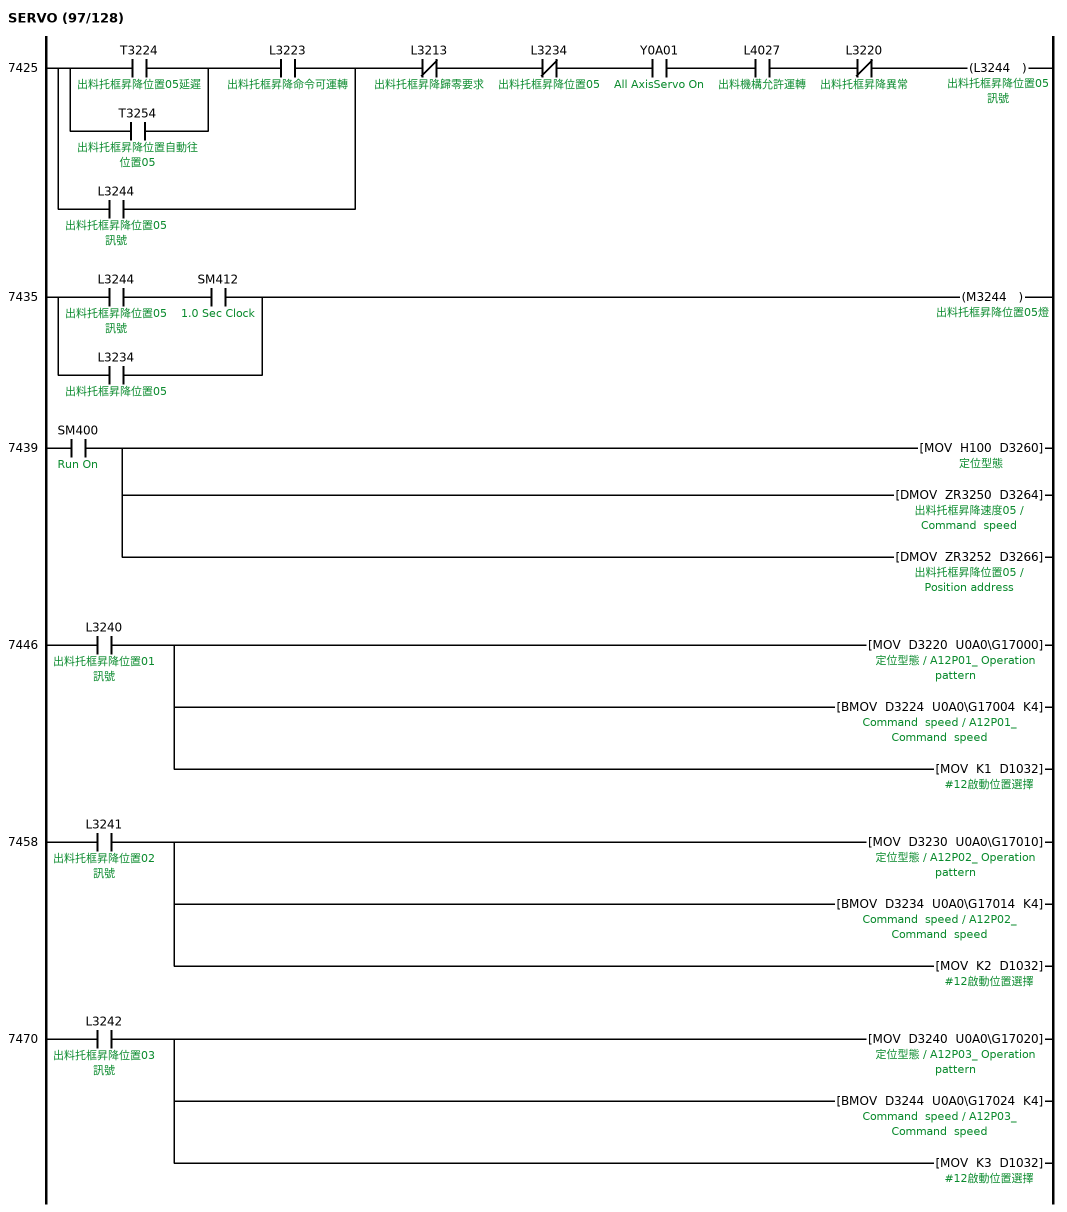
[picture p96: ladder of SERVO, rungs at steps 7425 to 7470]
7425  LD      T3224  ; 出料托框昇降位置05延遲
      OR      T3254  ; 出料托框昇降位置自動往  位置05
      AND     L3223  ; 出料托框昇降命令可運轉
      OR      L3244  ; 出料托框昇降位置05 訊號
      ANI     L3213  ; 出料托框昇降歸零要求
      ANI     L3234  ; 出料托框昇降位置05
      AND     Y0A01  ; All AxisServo On
      AND     L4027  ; 出料機構允許運轉
      ANI     L3220  ; 出料托框昇降異常
      OUT     L3244  ; 出料托框昇降位置05 訊號
7435  LD      L3244  ; 出料托框昇降位置05 訊號
      AND     SM412  ; 1.0 Sec Clock
      OR      L3234  ; 出料托框昇降位置05
      OUT     M3244  ; 出料托框昇降位置05燈
7439  LD      SM400  ; Run On
      MOV     H100 D3260  ; 定位型態
      DMOV    ZR3250 D3264  ; 出料托框昇降速度05 / Command  speed
      DMOV    ZR3252 D3266  ; Position address
7446  LD      L3240  ; 出料托框昇降位置01 訊號
      MOV     D3220 U0A0\G17000  ; A12P01_ Operation pattern
      BMOV    D3224 U0A0\G17004 K4  ; A12P01_ Command  speed
      MOV     K1 D1032  ; #12啟動位置選擇
7458  LD      L3241  ; 出料托框昇降位置02 訊號
      MOV     D3230 U0A0\G17010  ; A12P02_ Operation pattern
      BMOV    D3234 U0A0\G17014 K4  ; A12P02_ Command  speed
      MOV     K2 D1032
7470  LD      L3242  ; 出料托框昇降位置03 訊號
      MOV     D3240 U0A0\G17020  ; A12P03_ Operation pattern
      BMOV    D3244 U0A0\G17024 K4  ; A12P03_ Command  speed
      MOV     K3 D1032
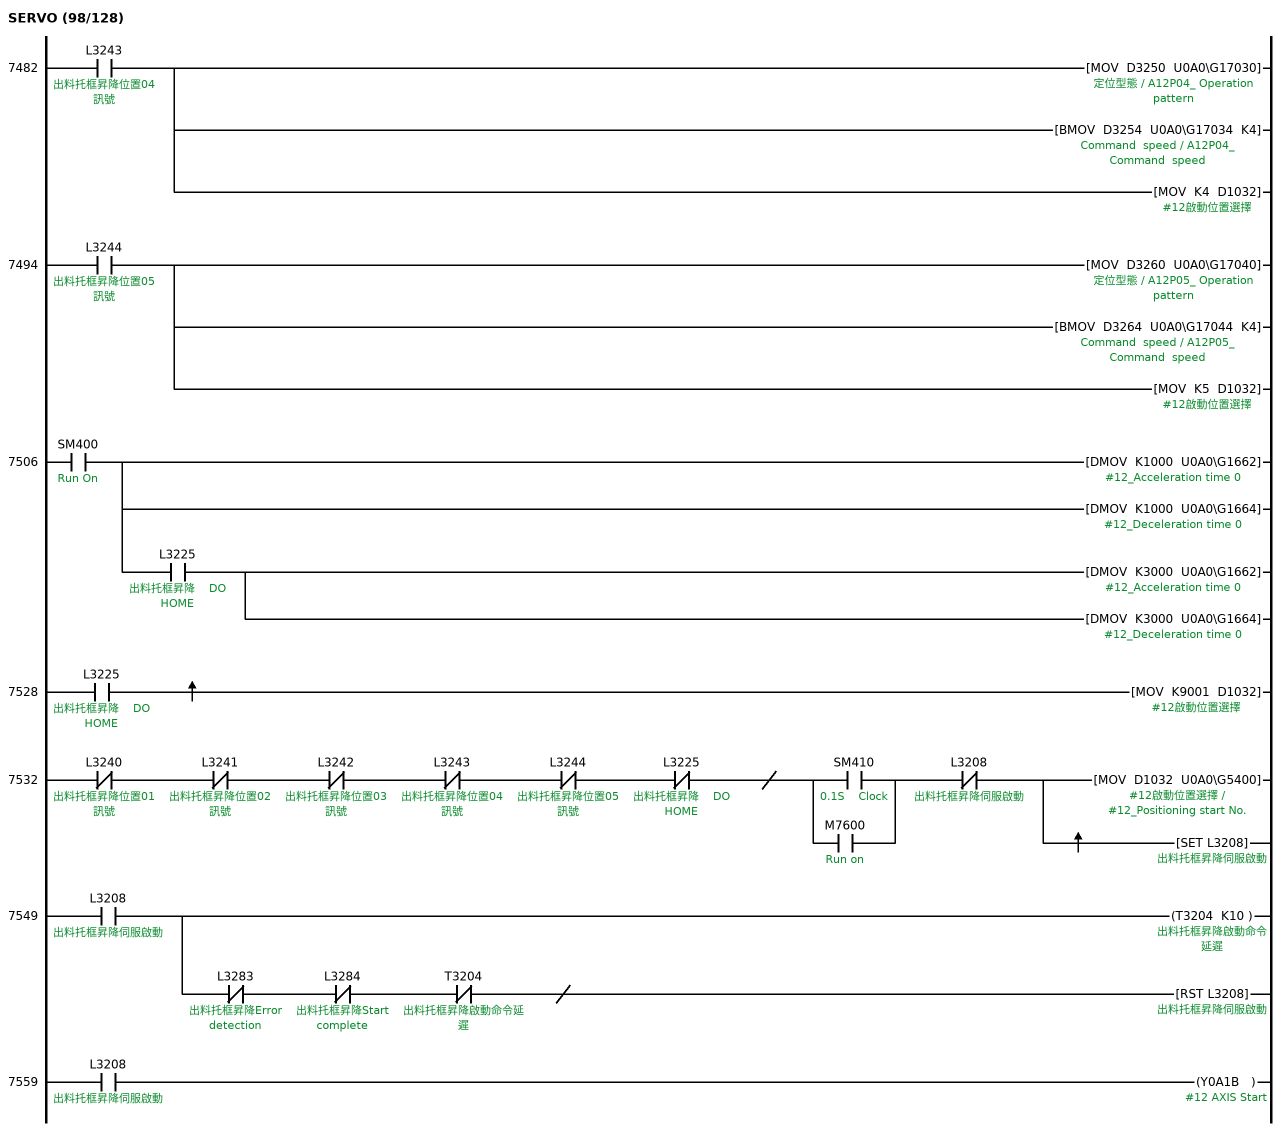
7482  LD      L3243  ; 出料托框昇降位置04 訊號
      MOV     D3250 U0A0\G17030  ; A12P04_ Operation pattern
      BMOV    D3254 U0A0\G17034 K4  ; A12P04_ Command  speed
      MOV     K4 D1032
7494  LD      L3244  ; 出料托框昇降位置05 訊號
      MOV     D3260 U0A0\G17040  ; A12P05_ Operation pattern
      BMOV    D3264 U0A0\G17044 K4  ; A12P05_ Command  speed
      MOV     K5 D1032
7506  LD      SM400  ; Run On
      DMOV    K1000 U0A0\G1662  ; #12_Acceleration time 0
      DMOV    K1000 U0A0\G1664  ; #12_Deceleration time 0
      AND     L3225  ; 出料托框昇降    DO HOME
      DMOV    K3000 U0A0\G1662
      DMOV    K3000 U0A0\G1664
7528  LD      L3225  ; 出料托框昇降    DO HOME
      MEP
      MOV     K9001 D1032
7532  LDI     L3240  ; 出料托框昇降位置01 訊號
      ANI     L3241  ; 出料托框昇降位置02 訊號
      ANI     L3242  ; 出料托框昇降位置03 訊號
      ANI     L3243  ; 出料托框昇降位置04 訊號
      ANI     L3244  ; 出料托框昇降位置05 訊號
      ANI     L3225  ; 出料托框昇降    DO HOME
      INV
      LD      SM410  ; 0.1S    Clock
      OR      M7600  ; Run on
      ANB
      ANI     L3208  ; 出料托框昇降伺服啟動
      MOV     D1032 U0A0\G5400  ; #12_Positioning start No.
      MEP
      SET     L3208  ; 出料托框昇降伺服啟動
7549  LD      L3208  ; 出料托框昇降伺服啟動
      OUT     T3204 K10  ; 出料托框昇降啟動命令延遲
      ANI     L3283  ; 出料托框昇降Error detection
      ANI     L3284  ; 出料托框昇降Start complete
      ANI     T3204  ; 出料托框昇降啟動命令延遲
      INV
      RST     L3208  ; 出料托框昇降伺服啟動
7559  LD      L3208  ; 出料托框昇降伺服啟動
      OUT     Y0A1B  ; #12 AXIS Start
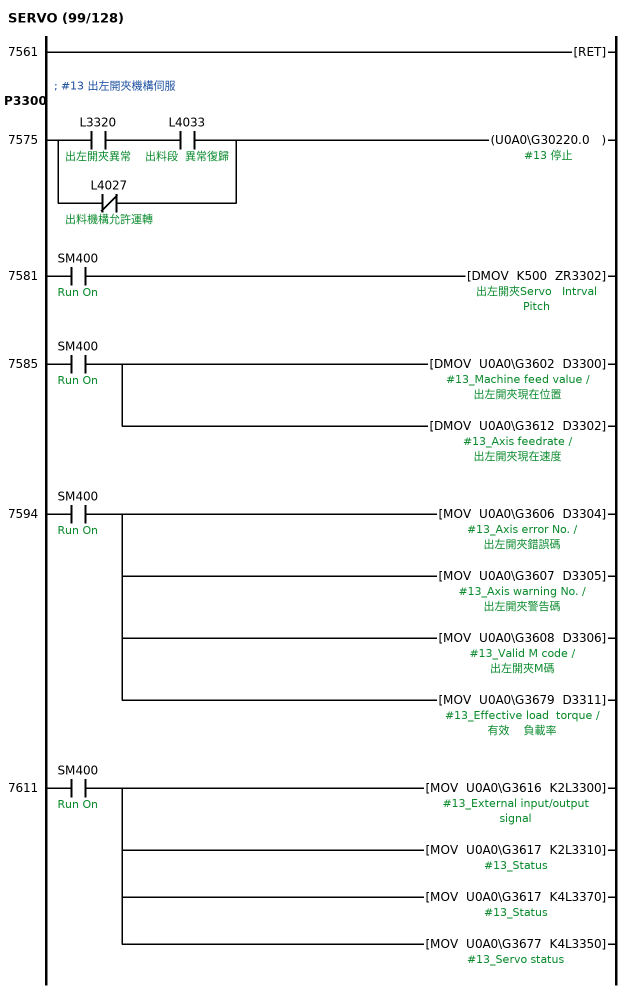
7561  RET
; #13 出左開夾機構伺服
      P3300
7575  LD      L3320  ; 出左開夾異常
      AND     L4033  ; 出料段  異常復歸
      ORI     L4027  ; 出料機構允許運轉
      OUT     U0A0\G30220.0  ; #13 停止
7581  LD      SM400  ; Run On
      DMOV    K500 ZR3302  ; 出左開夾Servo   Intrval Pitch
7585  LD      SM400  ; Run On
      DMOV    U0A0\G3602 D3300  ; #13_Machine feed value / 出左開夾現在位置
      DMOV    U0A0\G3612 D3302  ; #13_Axis feedrate / 出左開夾現在速度
7594  LD      SM400  ; Run On
      MOV     U0A0\G3606 D3304  ; #13_Axis error No. / 出左開夾錯誤碼
      MOV     U0A0\G3607 D3305  ; #13_Axis warning No. / 出左開夾警告碼
      MOV     U0A0\G3608 D3306  ; #13_Valid M code / 出左開夾M碼
      MOV     U0A0\G3679 D3311  ; #13_Effective load  torque / 有效    負載率
7611  LD      SM400  ; Run On
      MOV     U0A0\G3616 K2L3300  ; #13_External input/output signal / 出左開夾    負極限
      MOV     U0A0\G3617 K2L3310  ; #13_Status / 出左開夾速度控制
      MOV     U0A0\G3617 K4L3370  ; 出左開夾速度控制
      MOV     U0A0\G3677 K4L3350  ; #13_Servo status / READY ON
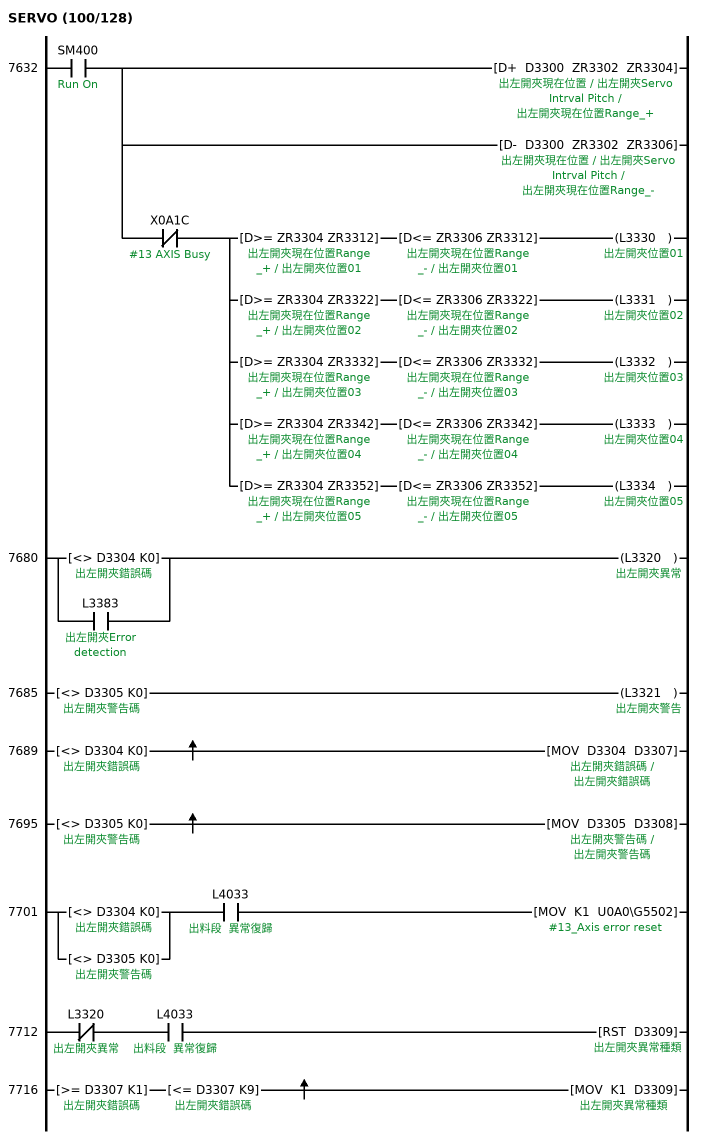
7632  LD      SM400  ; Run On
      D+      D3300 ZR3302 ZR3304  ; 出左開夾現在位置Range_+
      D-      D3300 ZR3302 ZR3306  ; 出左開夾現在位置Range_-
      ANI     X0A1C  ; #13 AXIS Busy
      MPS
      ANDD>=  ZR3304 ZR3312  ; 出左開夾現在位置Range_+ / 出左開夾位置01
      ANDD<=  ZR3306 ZR3312  ; 出左開夾現在位置Range_- / 出左開夾位置01
      OUT     L3330  ; 出左開夾位置01
      MRD
      ANDD>=  ZR3304 ZR3322  ; 出左開夾現在位置Range_+ / 出左開夾位置02
      ANDD<=  ZR3306 ZR3322  ; 出左開夾現在位置Range_- / 出左開夾位置02
      OUT     L3331  ; 出左開夾位置02
      MRD
      ANDD>=  ZR3304 ZR3332  ; 出左開夾現在位置Range_+ / 出左開夾位置03
      ANDD<=  ZR3306 ZR3332  ; 出左開夾現在位置Range_- / 出左開夾位置03
      OUT     L3332  ; 出左開夾位置03
      MRD
      ANDD>=  ZR3304 ZR3342  ; 出左開夾現在位置Range_+ / 出左開夾位置04
      ANDD<=  ZR3306 ZR3342  ; 出左開夾現在位置Range_- / 出左開夾位置04
      OUT     L3333  ; 出左開夾位置04
      MPP
      ANDD>=  ZR3304 ZR3352  ; 出左開夾現在位置Range_+ / 出左開夾位置05
      ANDD<=  ZR3306 ZR3352  ; 出左開夾現在位置Range_- / 出左開夾位置05
      OUT     L3334  ; 出左開夾位置05
7680  LD<>    D3304 K0  ; 出左開夾錯誤碼
      OR      L3383  ; 出左開夾Error detection
      OUT     L3320  ; 出左開夾異常
7685  LD<>    D3305 K0  ; 出左開夾警告碼
      OUT     L3321  ; 出左開夾警告
7689  LD<>    D3304 K0  ; 出左開夾錯誤碼
      MEP
      MOV     D3304 D3307  ; 出左開夾錯誤碼
7695  LD<>    D3305 K0  ; 出左開夾警告碼
      MEP
      MOV     D3305 D3308  ; 出左開夾警告碼
7701  LD<>    D3304 K0  ; 出左開夾錯誤碼
      OR<>    D3305 K0  ; 出左開夾警告碼
      AND     L4033  ; 出料段  異常復歸
      MOV     K1 U0A0\G5502  ; #13_Axis error reset
7712  LDI     L3320  ; 出左開夾異常
      AND     L4033  ; 出料段  異常復歸
      RST     D3309  ; 出左開夾異常種類
7716  LD>=    D3307 K1  ; 出左開夾錯誤碼
      AND<=   D3307 K9  ; 出左開夾錯誤碼
      MEP
      MOV     K1 D3309
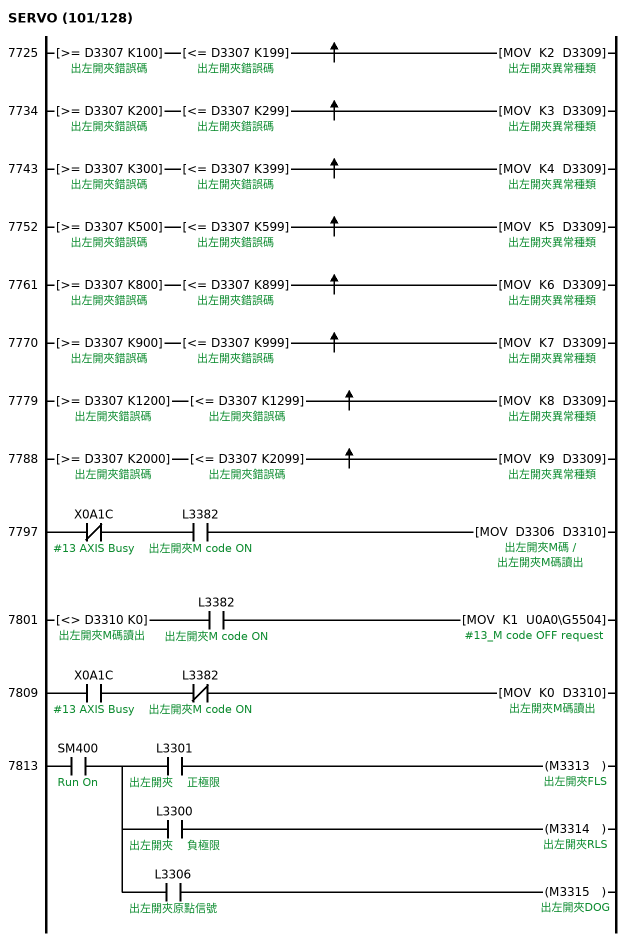
7725  LD>=    D3307 K100  ; 出左開夾錯誤碼
      AND<=   D3307 K199  ; 出左開夾錯誤碼
      MEP
      MOV     K2 D3309
7734  LD>=    D3307 K200  ; 出左開夾錯誤碼
      AND<=   D3307 K299  ; 出左開夾錯誤碼
      MEP
      MOV     K3 D3309
7743  LD>=    D3307 K300  ; 出左開夾錯誤碼
      AND<=   D3307 K399  ; 出左開夾錯誤碼
      MEP
      MOV     K4 D3309
7752  LD>=    D3307 K500  ; 出左開夾錯誤碼
      AND<=   D3307 K599  ; 出左開夾錯誤碼
      MEP
      MOV     K5 D3309
7761  LD>=    D3307 K800  ; 出左開夾錯誤碼
      AND<=   D3307 K899  ; 出左開夾錯誤碼
      MEP
      MOV     K6 D3309
7770  LD>=    D3307 K900  ; 出左開夾錯誤碼
      AND<=   D3307 K999  ; 出左開夾錯誤碼
      MEP
      MOV     K7 D3309
7779  LD>=    D3307 K1200  ; 出左開夾錯誤碼
      AND<=   D3307 K1299  ; 出左開夾錯誤碼
      MEP
      MOV     K8 D3309
7788  LD>=    D3307 K2000  ; 出左開夾錯誤碼
      AND<=   D3307 K2099  ; 出左開夾錯誤碼
      MEP
      MOV     K9 D3309
7797  LDI     X0A1C  ; #13 AXIS Busy
      AND     L3382  ; 出左開夾M code ON
      MOV     D3306 D3310  ; 出左開夾M碼讀出
7801  LD<>    D3310 K0  ; 出左開夾M碼讀出
      AND     L3382  ; 出左開夾M code ON
      MOV     K1 U0A0\G5504  ; #13_M code OFF request
7809  LD      X0A1C  ; #13 AXIS Busy
      ANI     L3382  ; 出左開夾M code ON
      MOV     K0 D3310
7813  LD      SM400  ; Run On
      MPS
      AND     L3301  ; 出左開夾    正極限
      OUT     M3313  ; 出左開夾FLS
      MRD
      AND     L3300  ; 出左開夾    負極限
      OUT     M3314  ; 出左開夾RLS
      MPP
      AND     L3306  ; 出左開夾原點信號
      OUT     M3315  ; 出左開夾DOG
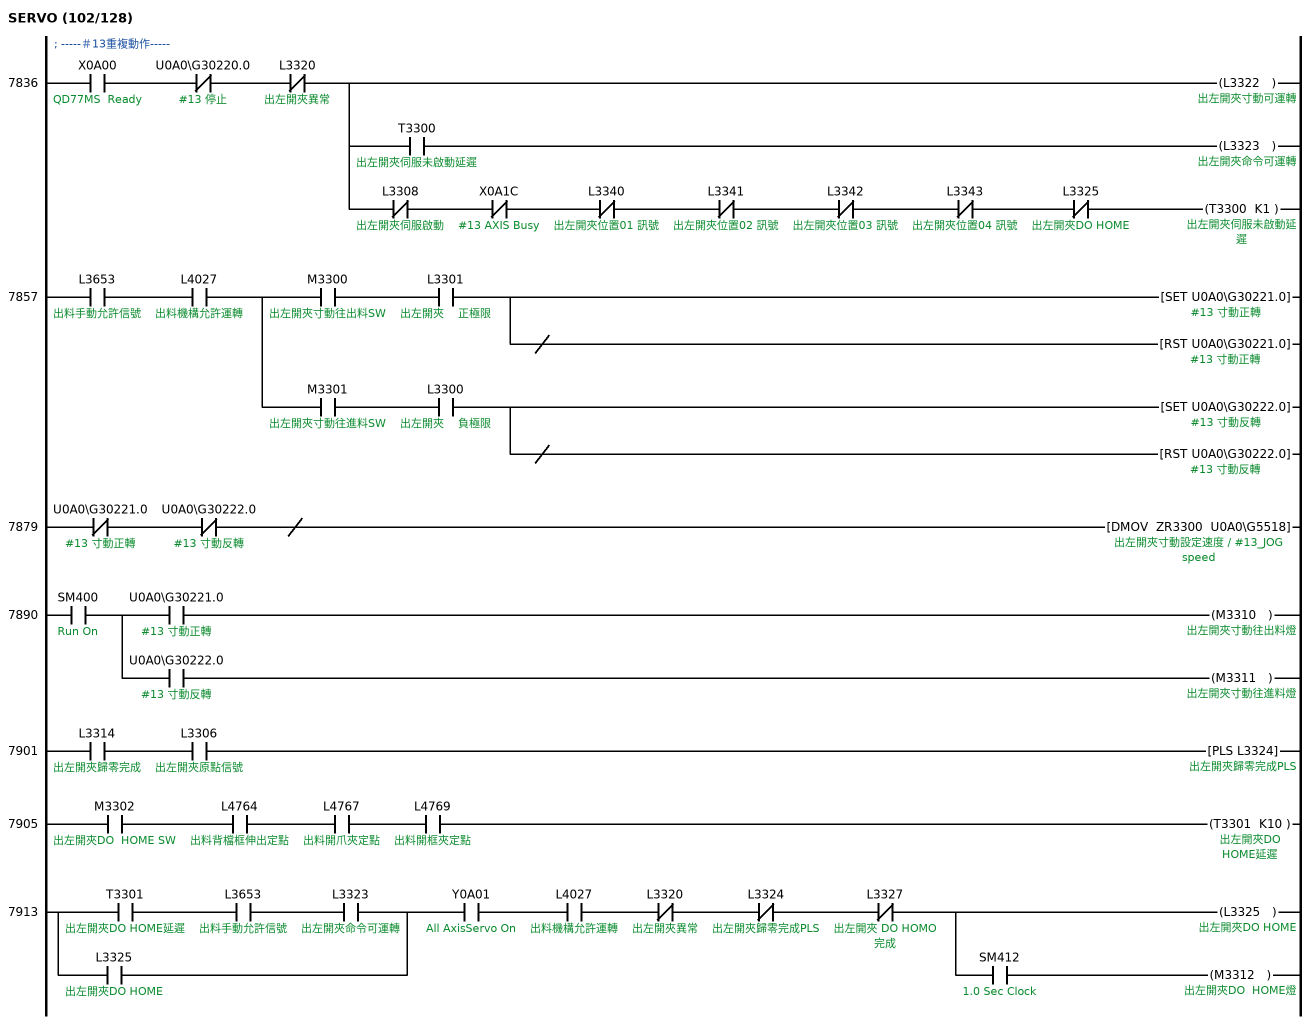
; -----＃13重複動作-----
7836  LD      X0A00  ; QD77MS  Ready
      ANI     U0A0\G30220.0  ; #13 停止
      ANI     L3320  ; 出左開夾異常
      OUT     L3322  ; 出左開夾寸動可運轉
      MPS
      AND     T3300  ; 出左開夾伺服未啟動延遲
      OUT     L3323  ; 出左開夾命令可運轉
      MPP
      ANI     L3308  ; 出左開夾伺服啟動
      ANI     X0A1C  ; #13 AXIS Busy
      ANI     L3340  ; 出左開夾位置01 訊號
      ANI     L3341  ; 出左開夾位置02 訊號
      ANI     L3342  ; 出左開夾位置03 訊號
      ANI     L3343  ; 出左開夾位置04 訊號
      ANI     L3325  ; 出左開夾DO HOME
      OUT     T3300 K1  ; 出左開夾伺服未啟動延遲
7857  LD      L3653  ; 出料手動允許信號
      AND     L4027  ; 出料機構允許運轉
      MPS
      AND     M3300  ; 出左開夾寸動往出料SW
      AND     L3301  ; 出左開夾    正極限
      SET     U0A0\G30221.0  ; #13 寸動正轉
      INV
      RST     U0A0\G30221.0  ; #13 寸動正轉
      MPP
      AND     M3301  ; 出左開夾寸動往進料SW
      AND     L3300  ; 出左開夾    負極限
      SET     U0A0\G30222.0  ; #13 寸動反轉
      INV
      RST     U0A0\G30222.0  ; #13 寸動反轉
7879  LDI     U0A0\G30221.0  ; #13 寸動正轉
      ANI     U0A0\G30222.0  ; #13 寸動反轉
      INV
      DMOV    ZR3300 U0A0\G5518  ; 出左開夾寸動設定速度 / #13_JOG     speed
7890  LD      SM400  ; Run On
      MPS
      AND     U0A0\G30221.0  ; #13 寸動正轉
      OUT     M3310  ; 出左開夾寸動往出料燈
      MPP
      AND     U0A0\G30222.0  ; #13 寸動反轉
      OUT     M3311  ; 出左開夾寸動往進料燈
7901  LD      L3314  ; 出左開夾歸零完成
      AND     L3306  ; 出左開夾原點信號
      PLS     L3324  ; 出左開夾歸零完成PLS
7905  LD      M3302  ; 出左開夾DO  HOME SW
      AND     L4764  ; 出料背檔框伸出定點
      AND     L4767  ; 出料開爪夾定點
      AND     L4769  ; 出料開框夾定點
      OUT     T3301 K10  ; 出左開夾DO HOME延遲
7913  LD      T3301  ; 出左開夾DO HOME延遲
      AND     L3653  ; 出料手動允許信號
      AND     L3323  ; 出左開夾命令可運轉
      OR      L3325  ; 出左開夾DO HOME
      AND     Y0A01  ; All AxisServo On
      AND     L4027  ; 出料機構允許運轉
      ANI     L3320  ; 出左開夾異常
      ANI     L3324  ; 出左開夾歸零完成PLS
      ANI     L3327  ; 出左開夾 DO HOMO 完成
      OUT     L3325  ; 出左開夾DO HOME
      AND     SM412  ; 1.0 Sec Clock
      OUT     M3312  ; 出左開夾DO  HOME燈
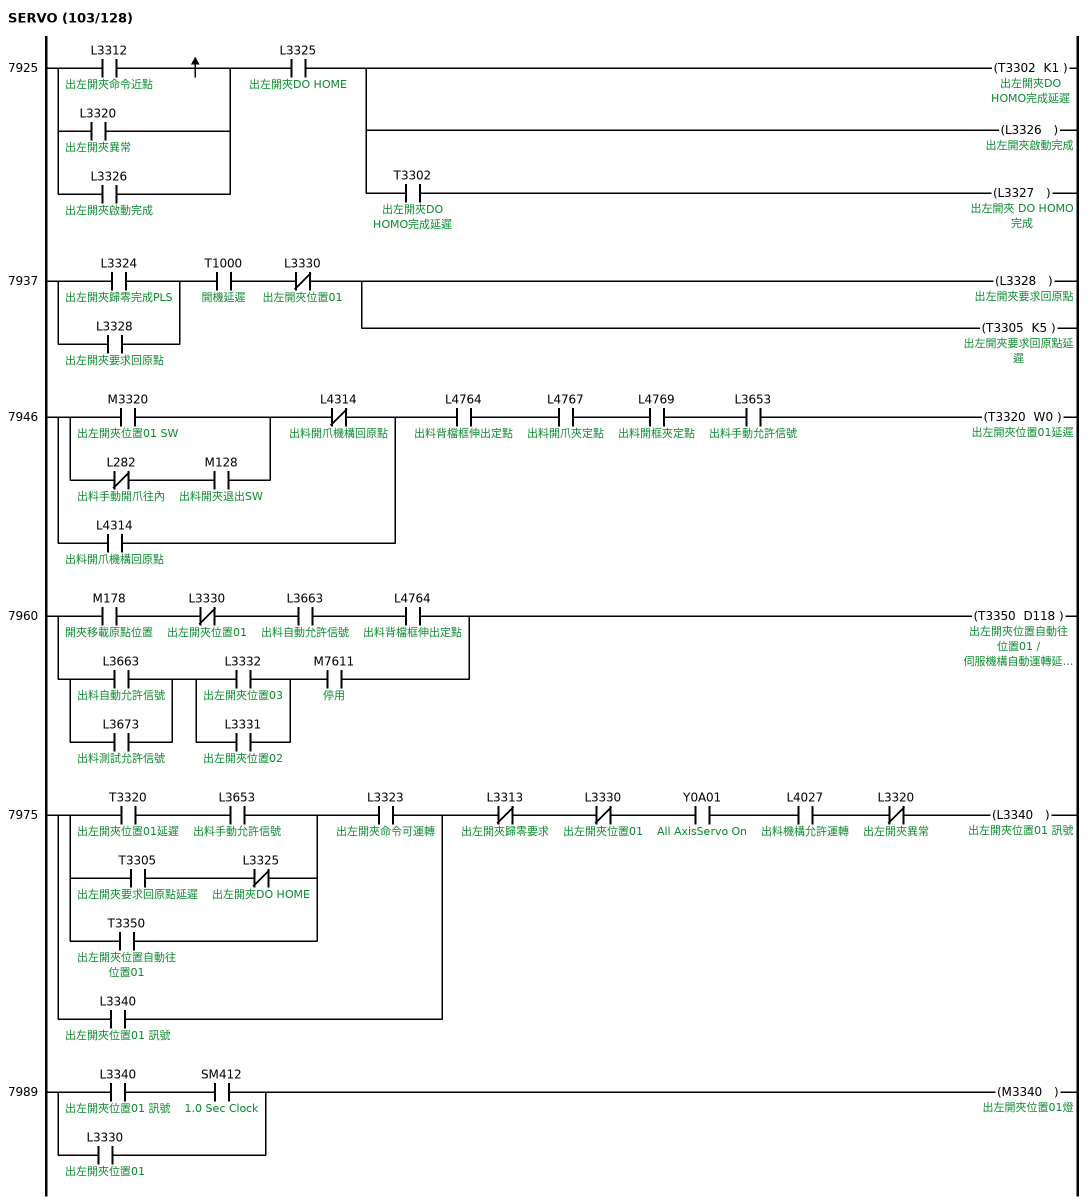
7925  LD      L3312  ; 出左開夾命令近點
      MEP
      OR      L3320  ; 出左開夾異常
      OR      L3326  ; 出左開夾啟動完成
      AND     L3325  ; 出左開夾DO HOME
      OUT     T3302 K1  ; 出左開夾DO HOMO完成延遲
      OUT     L3326  ; 出左開夾啟動完成
      AND     T3302  ; 出左開夾DO HOMO完成延遲
      OUT     L3327  ; 出左開夾 DO HOMO 完成
7937  LD      L3324  ; 出左開夾歸零完成PLS
      OR      L3328  ; 出左開夾要求回原點
      AND     T1000  ; 開機延遲
      ANI     L3330  ; 出左開夾位置01
      OUT     L3328  ; 出左開夾要求回原點
      OUT     T3305 K5  ; 出左開夾要求回原點延遲
7946  LD      M3320  ; 出左開夾位置01 SW
      LDI     L282  ; 出料手動開爪往內
      AND     M128  ; 出料開夾退出SW
      ORB
      ANI     L4314  ; 出料開爪機構回原點
      OR      L4314  ; 出料開爪機構回原點
      AND     L4764  ; 出料背檔框伸出定點
      AND     L4767  ; 出料開爪夾定點
      AND     L4769  ; 出料開框夾定點
      AND     L3653  ; 出料手動允許信號
      OUT     T3320 W0  ; 出左開夾位置01延遲
7960  LD      M178  ; 開夾移載原點位置
      ANI     L3330  ; 出左開夾位置01
      AND     L3663  ; 出料自動允許信號
      AND     L4764  ; 出料背檔框伸出定點
      LD      L3663  ; 出料自動允許信號
      OR      L3673  ; 出料測試允許信號
      LD      L3332  ; 出左開夾位置03
      OR      L3331  ; 出左開夾位置02
      ANB
      AND     M7611  ; 停用
      ORB
      OUT     T3350 D118  ; 出左開夾位置自動往  位置01 / 伺服機構自動運轉延遲時間
7975  LD      T3320  ; 出左開夾位置01延遲
      AND     L3653  ; 出料手動允許信號
      LD      T3305  ; 出左開夾要求回原點延遲
      ANI     L3325  ; 出左開夾DO HOME
      ORB
      OR      T3350  ; 出左開夾位置自動往  位置01
      AND     L3323  ; 出左開夾命令可運轉
      OR      L3340  ; 出左開夾位置01 訊號
      ANI     L3313  ; 出左開夾歸零要求
      ANI     L3330  ; 出左開夾位置01
      AND     Y0A01  ; All AxisServo On
      AND     L4027  ; 出料機構允許運轉
      ANI     L3320  ; 出左開夾異常
      OUT     L3340  ; 出左開夾位置01 訊號
7989  LD      L3340  ; 出左開夾位置01 訊號
      AND     SM412  ; 1.0 Sec Clock
      OR      L3330  ; 出左開夾位置01
      OUT     M3340  ; 出左開夾位置01燈
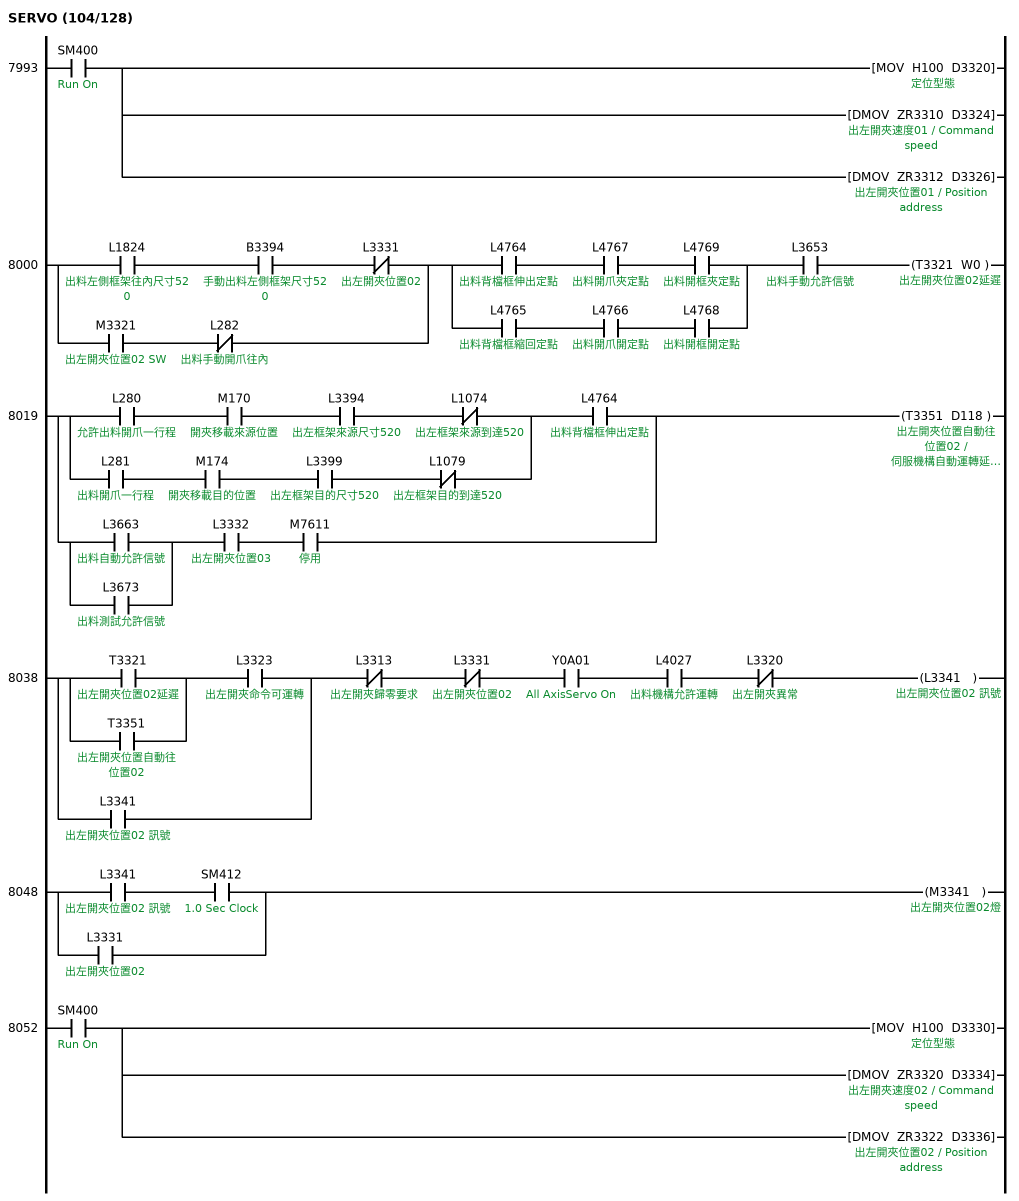
7993  LD      SM400  ; Run On
      MOV     H100 D3320  ; 定位型態
      DMOV    ZR3310 D3324  ; 出左開夾速度01 / Command  speed
      DMOV    ZR3312 D3326  ; Position address
8000  LD      L1824  ; 出料左側框架往內尺寸520
      AND     B3394  ; 手動出料左側框架尺寸520
      ANI     L3331  ; 出左開夾位置02
      LD      M3321  ; 出左開夾位置02 SW
      ANI     L282  ; 出料手動開爪往內
      ORB
      LD      L4764  ; 出料背檔框伸出定點
      AND     L4767  ; 出料開爪夾定點
      AND     L4769  ; 出料開框夾定點
      LD      L4765  ; 出料背檔框縮回定點
      AND     L4766  ; 出料開爪開定點
      AND     L4768  ; 出料開框開定點
      ORB
      ANB
      AND     L3653  ; 出料手動允許信號
      OUT     T3321 W0  ; 出左開夾位置02延遲
8019  LD      L280  ; 允許出料開爪一行程
      AND     M170  ; 開夾移載來源位置
      AND     L3394  ; 出左框架來源尺寸520
      ANI     L1074  ; 出左框架來源到達520
      LD      L281  ; 出料開爪一行程
      AND     M174  ; 開夾移載目的位置
      AND     L3399  ; 出左框架目的尺寸520
      ANI     L1079  ; 出左框架目的到達520
      ORB
      AND     L4764  ; 出料背檔框伸出定點
      LD      L3663  ; 出料自動允許信號
      OR      L3673  ; 出料測試允許信號
      AND     L3332  ; 出左開夾位置03
      AND     M7611  ; 停用
      ORB
      OUT     T3351 D118  ; 出左開夾位置自動往  位置02 / 伺服機構自動運轉延遲時間
8038  LD      T3321  ; 出左開夾位置02延遲
      OR      T3351  ; 出左開夾位置自動往  位置02
      AND     L3323  ; 出左開夾命令可運轉
      OR      L3341  ; 出左開夾位置02 訊號
      ANI     L3313  ; 出左開夾歸零要求
      ANI     L3331  ; 出左開夾位置02
      AND     Y0A01  ; All AxisServo On
      AND     L4027  ; 出料機構允許運轉
      ANI     L3320  ; 出左開夾異常
      OUT     L3341  ; 出左開夾位置02 訊號
8048  LD      L3341  ; 出左開夾位置02 訊號
      AND     SM412  ; 1.0 Sec Clock
      OR      L3331  ; 出左開夾位置02
      OUT     M3341  ; 出左開夾位置02燈
8052  LD      SM400  ; Run On
      MOV     H100 D3330  ; 定位型態
      DMOV    ZR3320 D3334  ; 出左開夾速度02 / Command  speed
      DMOV    ZR3322 D3336  ; Position address
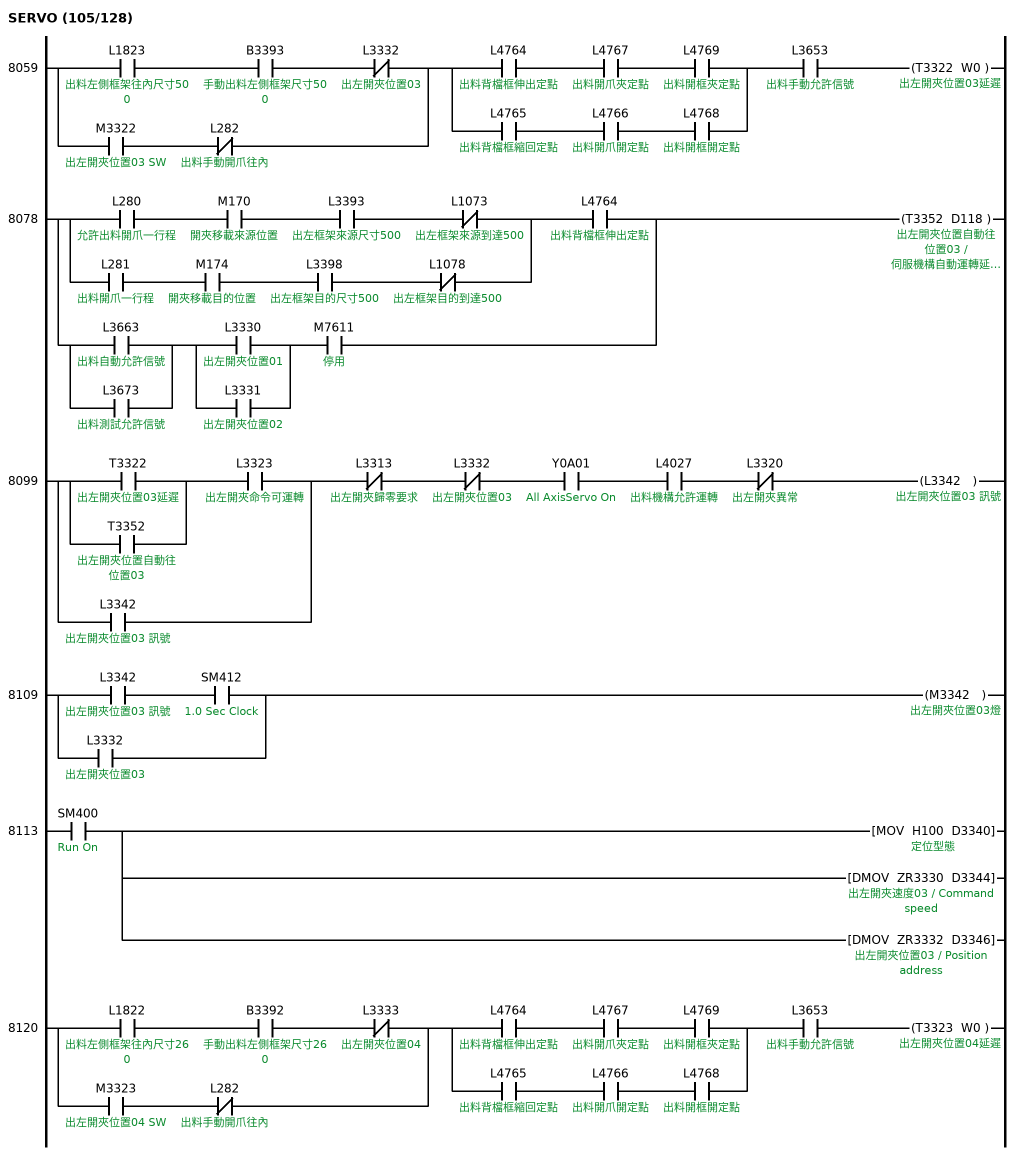
8059  LD      L1823  ; 出料左側框架往內尺寸500
      AND     B3393  ; 手動出料左側框架尺寸500
      ANI     L3332  ; 出左開夾位置03
      LD      M3322  ; 出左開夾位置03 SW
      ANI     L282  ; 出料手動開爪往內
      ORB
      LD      L4764  ; 出料背檔框伸出定點
      AND     L4767  ; 出料開爪夾定點
      AND     L4769  ; 出料開框夾定點
      LD      L4765  ; 出料背檔框縮回定點
      AND     L4766  ; 出料開爪開定點
      AND     L4768  ; 出料開框開定點
      ORB
      ANB
      AND     L3653  ; 出料手動允許信號
      OUT     T3322 W0  ; 出左開夾位置03延遲
8078  LD      L280  ; 允許出料開爪一行程
      AND     M170  ; 開夾移載來源位置
      AND     L3393  ; 出左框架來源尺寸500
      ANI     L1073  ; 出左框架來源到達500
      LD      L281  ; 出料開爪一行程
      AND     M174  ; 開夾移載目的位置
      AND     L3398  ; 出左框架目的尺寸500
      ANI     L1078  ; 出左框架目的到達500
      ORB
      AND     L4764  ; 出料背檔框伸出定點
      LD      L3663  ; 出料自動允許信號
      OR      L3673  ; 出料測試允許信號
      LD      L3330  ; 出左開夾位置01
      OR      L3331  ; 出左開夾位置02
      ANB
      AND     M7611  ; 停用
      ORB
      OUT     T3352 D118  ; 出左開夾位置自動往  位置03 / 伺服機構自動運轉延遲時間
8099  LD      T3322  ; 出左開夾位置03延遲
      OR      T3352  ; 出左開夾位置自動往  位置03
      AND     L3323  ; 出左開夾命令可運轉
      OR      L3342  ; 出左開夾位置03 訊號
      ANI     L3313  ; 出左開夾歸零要求
      ANI     L3332  ; 出左開夾位置03
      AND     Y0A01  ; All AxisServo On
      AND     L4027  ; 出料機構允許運轉
      ANI     L3320  ; 出左開夾異常
      OUT     L3342  ; 出左開夾位置03 訊號
8109  LD      L3342  ; 出左開夾位置03 訊號
      AND     SM412  ; 1.0 Sec Clock
      OR      L3332  ; 出左開夾位置03
      OUT     M3342  ; 出左開夾位置03燈
8113  LD      SM400  ; Run On
      MOV     H100 D3340  ; 定位型態
      DMOV    ZR3330 D3344  ; 出左開夾速度03 / Command  speed
      DMOV    ZR3332 D3346  ; Position address
8120  LD      L1822  ; 出料左側框架往內尺寸260
      AND     B3392  ; 手動出料左側框架尺寸260
      ANI     L3333  ; 出左開夾位置04
      LD      M3323  ; 出左開夾位置04 SW
      ANI     L282  ; 出料手動開爪往內
      ORB
      LD      L4764  ; 出料背檔框伸出定點
      AND     L4767  ; 出料開爪夾定點
      AND     L4769  ; 出料開框夾定點
      LD      L4765  ; 出料背檔框縮回定點
      AND     L4766  ; 出料開爪開定點
      AND     L4768  ; 出料開框開定點
      ORB
      ANB
      AND     L3653  ; 出料手動允許信號
      OUT     T3323 W0  ; 出左開夾位置04延遲
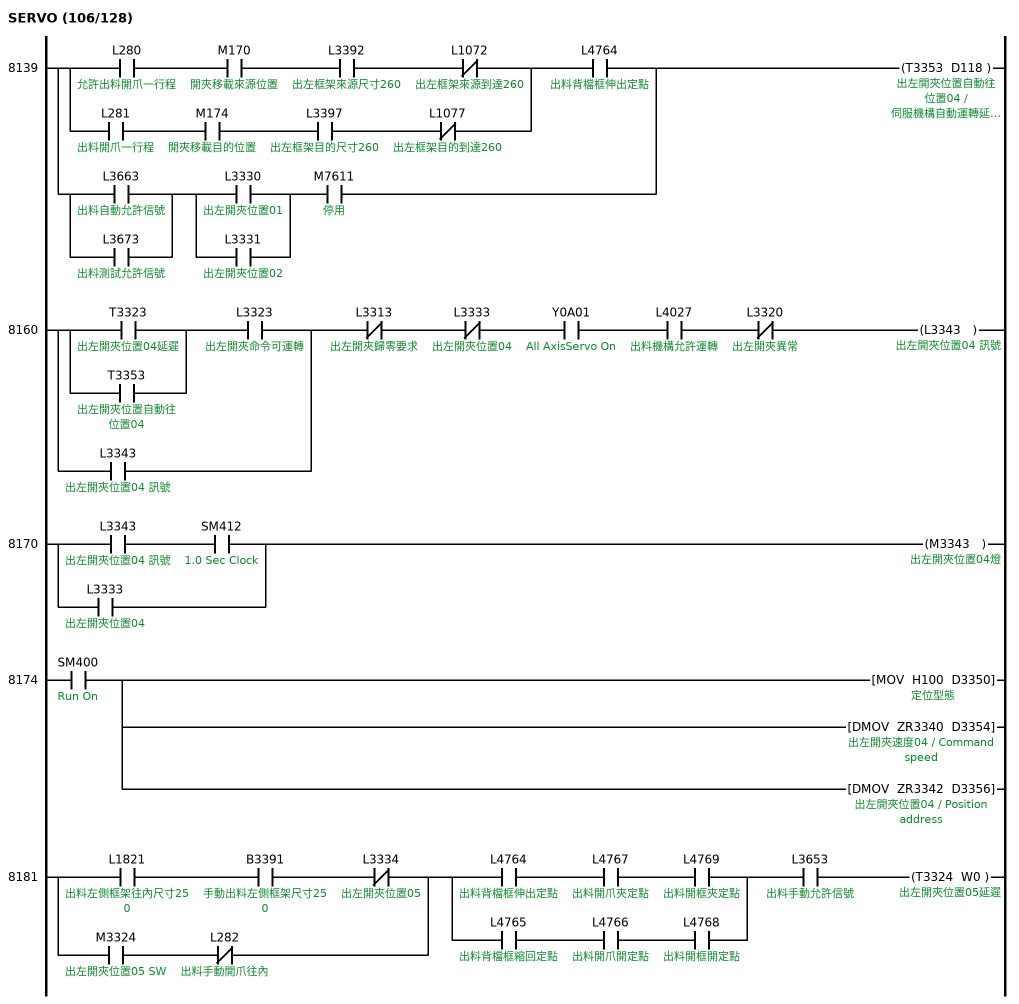
8139  LD      L280  ; 允許出料開爪一行程
      AND     M170  ; 開夾移載來源位置
      AND     L3392  ; 出左框架來源尺寸260
      ANI     L1072  ; 出左框架來源到達260
      LD      L281  ; 出料開爪一行程
      AND     M174  ; 開夾移載目的位置
      AND     L3397  ; 出左框架目的尺寸260
      ANI     L1077  ; 出左框架目的到達260
      ORB
      AND     L4764  ; 出料背檔框伸出定點
      LD      L3663  ; 出料自動允許信號
      OR      L3673  ; 出料測試允許信號
      LD      L3330  ; 出左開夾位置01
      OR      L3331  ; 出左開夾位置02
      ANB
      AND     M7611  ; 停用
      ORB
      OUT     T3353 D118  ; 出左開夾位置自動往  位置04 / 伺服機構自動運轉延遲時間
8160  LD      T3323  ; 出左開夾位置04延遲
      OR      T3353  ; 出左開夾位置自動往  位置04
      AND     L3323  ; 出左開夾命令可運轉
      OR      L3343  ; 出左開夾位置04 訊號
      ANI     L3313  ; 出左開夾歸零要求
      ANI     L3333  ; 出左開夾位置04
      AND     Y0A01  ; All AxisServo On
      AND     L4027  ; 出料機構允許運轉
      ANI     L3320  ; 出左開夾異常
      OUT     L3343  ; 出左開夾位置04 訊號
8170  LD      L3343  ; 出左開夾位置04 訊號
      AND     SM412  ; 1.0 Sec Clock
      OR      L3333  ; 出左開夾位置04
      OUT     M3343  ; 出左開夾位置04燈
8174  LD      SM400  ; Run On
      MOV     H100 D3350  ; 定位型態
      DMOV    ZR3340 D3354  ; 出左開夾速度04 / Command  speed
      DMOV    ZR3342 D3356  ; Position address
8181  LD      L1821  ; 出料左側框架往內尺寸250
      AND     B3391  ; 手動出料左側框架尺寸250
      ANI     L3334  ; 出左開夾位置05
      LD      M3324  ; 出左開夾位置05 SW
      ANI     L282  ; 出料手動開爪往內
      ORB
      LD      L4764  ; 出料背檔框伸出定點
      AND     L4767  ; 出料開爪夾定點
      AND     L4769  ; 出料開框夾定點
      LD      L4765  ; 出料背檔框縮回定點
      AND     L4766  ; 出料開爪開定點
      AND     L4768  ; 出料開框開定點
      ORB
      ANB
      AND     L3653  ; 出料手動允許信號
      OUT     T3324 W0  ; 出左開夾位置05延遲
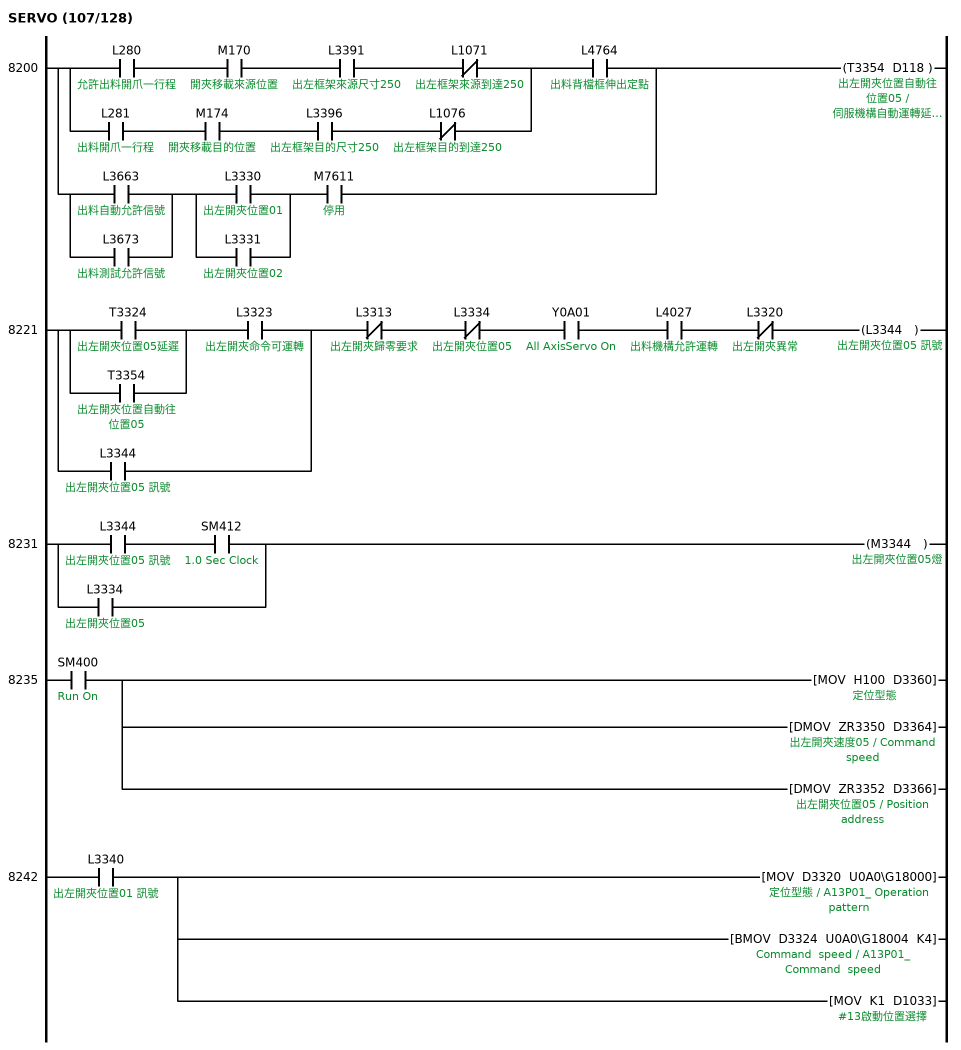
8200  LD      L280  ; 允許出料開爪一行程
      AND     M170  ; 開夾移載來源位置
      AND     L3391  ; 出左框架來源尺寸250
      ANI     L1071  ; 出左框架來源到達250
      LD      L281  ; 出料開爪一行程
      AND     M174  ; 開夾移載目的位置
      AND     L3396  ; 出左框架目的尺寸250
      ANI     L1076  ; 出左框架目的到達250
      ORB
      AND     L4764  ; 出料背檔框伸出定點
      LD      L3663  ; 出料自動允許信號
      OR      L3673  ; 出料測試允許信號
      LD      L3330  ; 出左開夾位置01
      OR      L3331  ; 出左開夾位置02
      ANB
      AND     M7611  ; 停用
      ORB
      OUT     T3354 D118  ; 出左開夾位置自動往  位置05 / 伺服機構自動運轉延遲時間
8221  LD      T3324  ; 出左開夾位置05延遲
      OR      T3354  ; 出左開夾位置自動往  位置05
      AND     L3323  ; 出左開夾命令可運轉
      OR      L3344  ; 出左開夾位置05 訊號
      ANI     L3313  ; 出左開夾歸零要求
      ANI     L3334  ; 出左開夾位置05
      AND     Y0A01  ; All AxisServo On
      AND     L4027  ; 出料機構允許運轉
      ANI     L3320  ; 出左開夾異常
      OUT     L3344  ; 出左開夾位置05 訊號
8231  LD      L3344  ; 出左開夾位置05 訊號
      AND     SM412  ; 1.0 Sec Clock
      OR      L3334  ; 出左開夾位置05
      OUT     M3344  ; 出左開夾位置05燈
8235  LD      SM400  ; Run On
      MOV     H100 D3360  ; 定位型態
      DMOV    ZR3350 D3364  ; 出左開夾速度05 / Command  speed
      DMOV    ZR3352 D3366  ; Position address
8242  LD      L3340  ; 出左開夾位置01 訊號
      MOV     D3320 U0A0\G18000  ; A13P01_ Operation pattern
      BMOV    D3324 U0A0\G18004 K4  ; A13P01_ Command  speed
      MOV     K1 D1033  ; #13啟動位置選擇
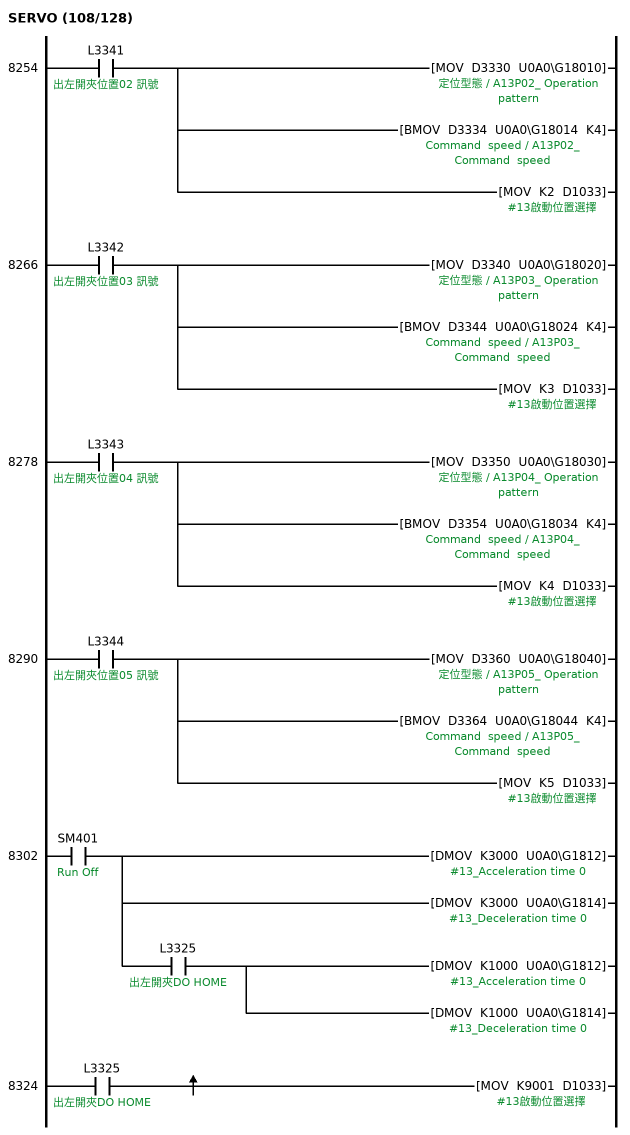
8254  LD      L3341  ; 出左開夾位置02 訊號
      MOV     D3330 U0A0\G18010  ; A13P02_ Operation pattern
      BMOV    D3334 U0A0\G18014 K4  ; A13P02_ Command  speed
      MOV     K2 D1033
8266  LD      L3342  ; 出左開夾位置03 訊號
      MOV     D3340 U0A0\G18020  ; A13P03_ Operation pattern
      BMOV    D3344 U0A0\G18024 K4  ; A13P03_ Command  speed
      MOV     K3 D1033
8278  LD      L3343  ; 出左開夾位置04 訊號
      MOV     D3350 U0A0\G18030  ; A13P04_ Operation pattern
      BMOV    D3354 U0A0\G18034 K4  ; A13P04_ Command  speed
      MOV     K4 D1033
8290  LD      L3344  ; 出左開夾位置05 訊號
      MOV     D3360 U0A0\G18040  ; A13P05_ Operation pattern
      BMOV    D3364 U0A0\G18044 K4  ; A13P05_ Command  speed
      MOV     K5 D1033
8302  LD      SM401  ; Run Off
      DMOV    K3000 U0A0\G1812  ; #13_Acceleration time 0
      DMOV    K3000 U0A0\G1814  ; #13_Deceleration time 0
      AND     L3325  ; 出左開夾DO HOME
      DMOV    K1000 U0A0\G1812
      DMOV    K1000 U0A0\G1814
8324  LD      L3325  ; 出左開夾DO HOME
      MEP
      MOV     K9001 D1033
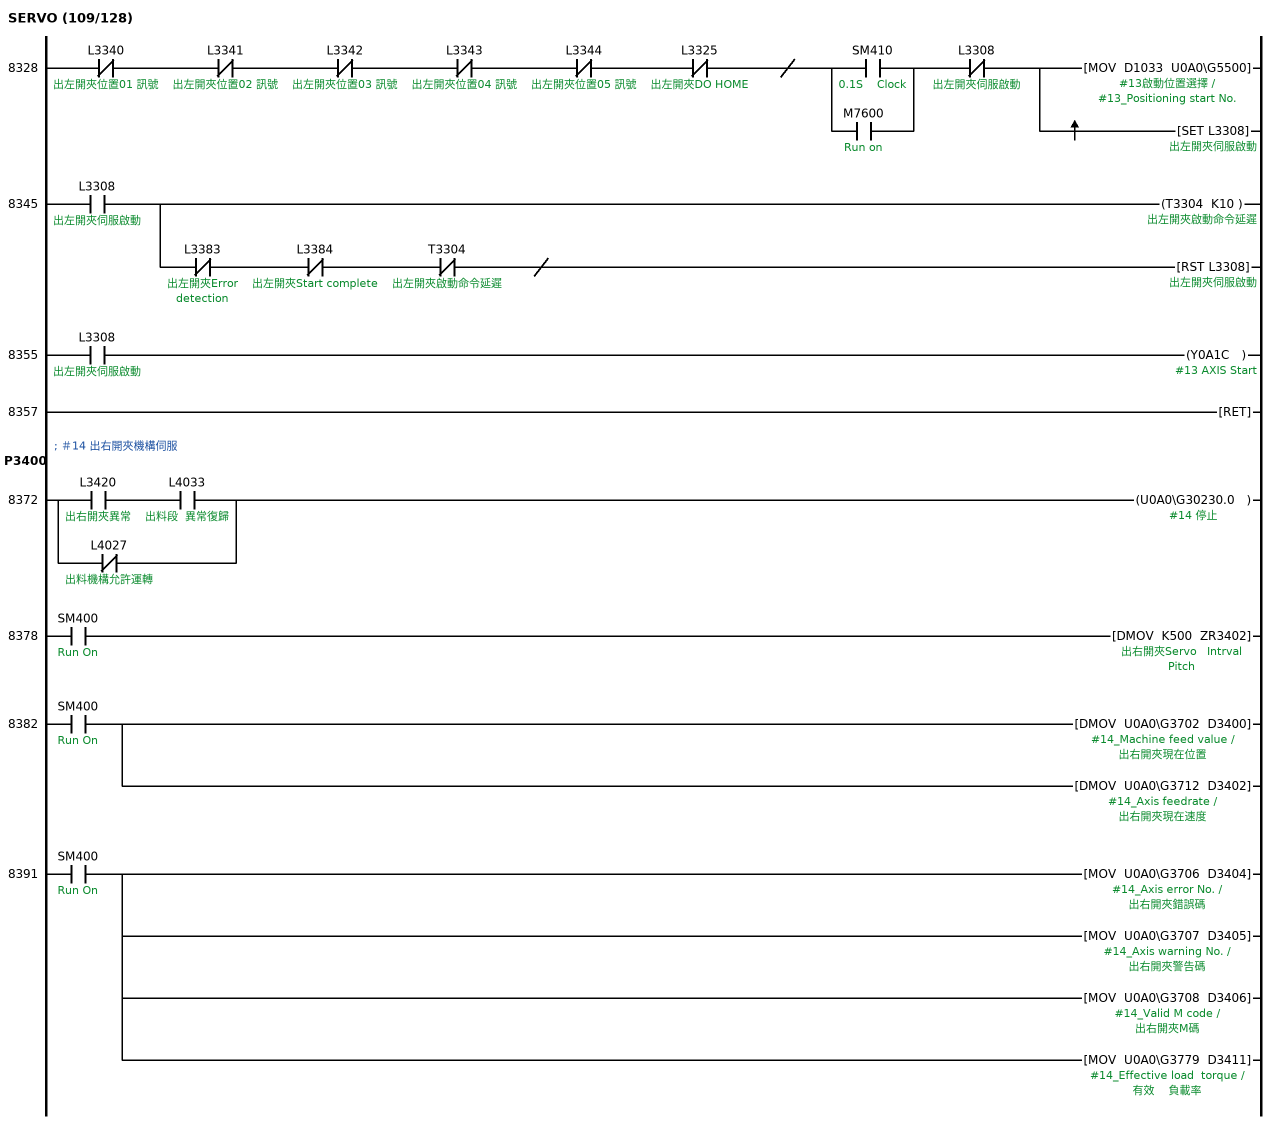
8328  LDI     L3340  ; 出左開夾位置01 訊號
      ANI     L3341  ; 出左開夾位置02 訊號
      ANI     L3342  ; 出左開夾位置03 訊號
      ANI     L3343  ; 出左開夾位置04 訊號
      ANI     L3344  ; 出左開夾位置05 訊號
      ANI     L3325  ; 出左開夾DO HOME
      INV
      LD      SM410  ; 0.1S    Clock
      OR      M7600  ; Run on
      ANB
      ANI     L3308  ; 出左開夾伺服啟動
      MOV     D1033 U0A0\G5500  ; #13_Positioning start No.
      MEP
      SET     L3308  ; 出左開夾伺服啟動
8345  LD      L3308  ; 出左開夾伺服啟動
      OUT     T3304 K10  ; 出左開夾啟動命令延遲
      ANI     L3383  ; 出左開夾Error detection
      ANI     L3384  ; 出左開夾Start complete
      ANI     T3304  ; 出左開夾啟動命令延遲
      INV
      RST     L3308  ; 出左開夾伺服啟動
8355  LD      L3308  ; 出左開夾伺服啟動
      OUT     Y0A1C  ; #13 AXIS Start
8357  RET
; ＃14 出右開夾機構伺服
      P3400
8372  LD      L3420  ; 出右開夾異常
      AND     L4033  ; 出料段  異常復歸
      ORI     L4027  ; 出料機構允許運轉
      OUT     U0A0\G30230.0  ; #14 停止
8378  LD      SM400  ; Run On
      DMOV    K500 ZR3402  ; 出右開夾Servo   Intrval Pitch
8382  LD      SM400  ; Run On
      DMOV    U0A0\G3702 D3400  ; #14_Machine feed value / 出右開夾現在位置
      DMOV    U0A0\G3712 D3402  ; #14_Axis feedrate / 出右開夾現在速度
8391  LD      SM400  ; Run On
      MOV     U0A0\G3706 D3404  ; #14_Axis error No. / 出右開夾錯誤碼
      MOV     U0A0\G3707 D3405  ; #14_Axis warning No. / 出右開夾警告碼
      MOV     U0A0\G3708 D3406  ; #14_Valid M code / 出右開夾M碼
      MOV     U0A0\G3779 D3411  ; #14_Effective load  torque / 有效    負載率
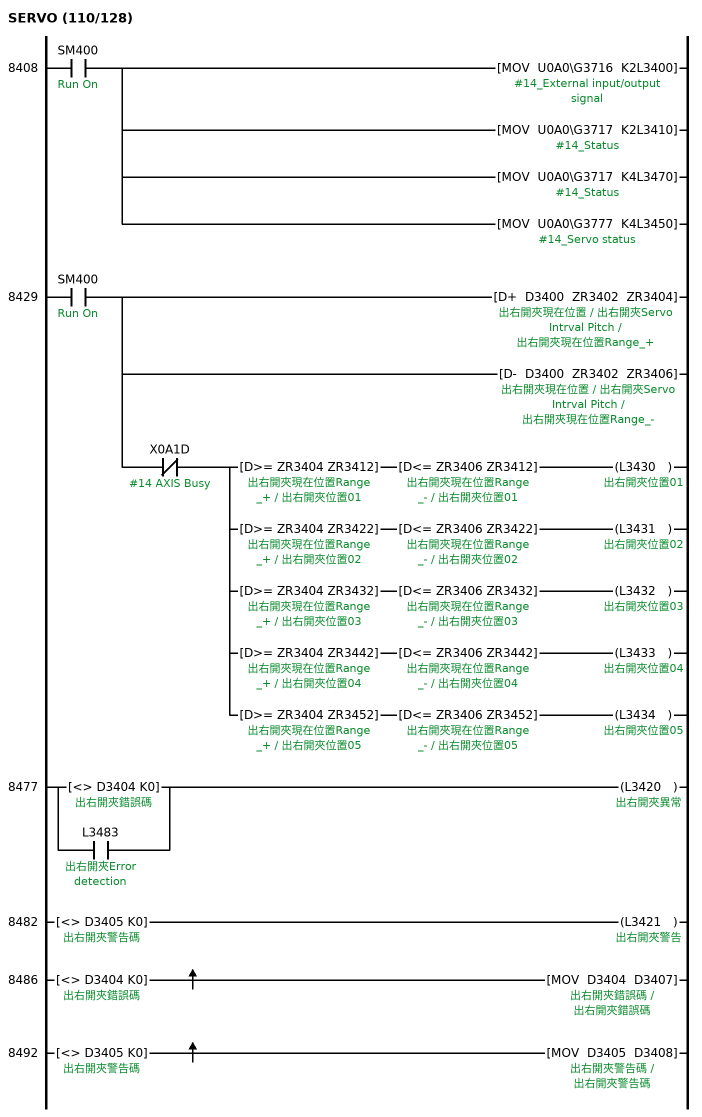
8408  LD      SM400  ; Run On
      MOV     U0A0\G3716 K2L3400  ; #14_External input/output signal / 出右開夾    負極限
      MOV     U0A0\G3717 K2L3410  ; #14_Status / 出右開夾速度控制
      MOV     U0A0\G3717 K4L3470  ; 出右開夾速度控制
      MOV     U0A0\G3777 K4L3450  ; #14_Servo status / READY ON
8429  LD      SM400  ; Run On
      D+      D3400 ZR3402 ZR3404  ; 出右開夾現在位置Range_+
      D-      D3400 ZR3402 ZR3406  ; 出右開夾現在位置Range_-
      ANI     X0A1D  ; #14 AXIS Busy
      MPS
      ANDD>=  ZR3404 ZR3412  ; 出右開夾現在位置Range_+ / 出右開夾位置01
      ANDD<=  ZR3406 ZR3412  ; 出右開夾現在位置Range_- / 出右開夾位置01
      OUT     L3430  ; 出右開夾位置01
      MRD
      ANDD>=  ZR3404 ZR3422  ; 出右開夾現在位置Range_+ / 出右開夾位置02
      ANDD<=  ZR3406 ZR3422  ; 出右開夾現在位置Range_- / 出右開夾位置02
      OUT     L3431  ; 出右開夾位置02
      MRD
      ANDD>=  ZR3404 ZR3432  ; 出右開夾現在位置Range_+ / 出右開夾位置03
      ANDD<=  ZR3406 ZR3432  ; 出右開夾現在位置Range_- / 出右開夾位置03
      OUT     L3432  ; 出右開夾位置03
      MRD
      ANDD>=  ZR3404 ZR3442  ; 出右開夾現在位置Range_+ / 出右開夾位置04
      ANDD<=  ZR3406 ZR3442  ; 出右開夾現在位置Range_- / 出右開夾位置04
      OUT     L3433  ; 出右開夾位置04
      MPP
      ANDD>=  ZR3404 ZR3452  ; 出右開夾現在位置Range_+ / 出右開夾位置05
      ANDD<=  ZR3406 ZR3452  ; 出右開夾現在位置Range_- / 出右開夾位置05
      OUT     L3434  ; 出右開夾位置05
8477  LD<>    D3404 K0  ; 出右開夾錯誤碼
      OR      L3483  ; 出右開夾Error detection
      OUT     L3420  ; 出右開夾異常
8482  LD<>    D3405 K0  ; 出右開夾警告碼
      OUT     L3421  ; 出右開夾警告
8486  LD<>    D3404 K0  ; 出右開夾錯誤碼
      MEP
      MOV     D3404 D3407  ; 出右開夾錯誤碼
8492  LD<>    D3405 K0  ; 出右開夾警告碼
      MEP
      MOV     D3405 D3408  ; 出右開夾警告碼
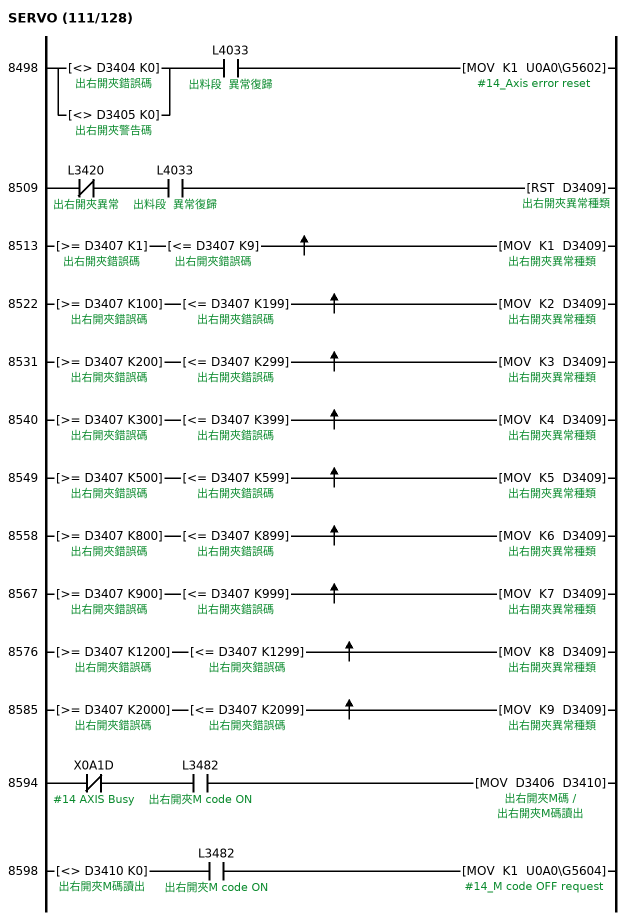
8498  LD<>    D3404 K0  ; 出右開夾錯誤碼
      OR<>    D3405 K0  ; 出右開夾警告碼
      AND     L4033  ; 出料段  異常復歸
      MOV     K1 U0A0\G5602  ; #14_Axis error reset
8509  LDI     L3420  ; 出右開夾異常
      AND     L4033  ; 出料段  異常復歸
      RST     D3409  ; 出右開夾異常種類
8513  LD>=    D3407 K1  ; 出右開夾錯誤碼
      AND<=   D3407 K9  ; 出右開夾錯誤碼
      MEP
      MOV     K1 D3409
8522  LD>=    D3407 K100  ; 出右開夾錯誤碼
      AND<=   D3407 K199  ; 出右開夾錯誤碼
      MEP
      MOV     K2 D3409
8531  LD>=    D3407 K200  ; 出右開夾錯誤碼
      AND<=   D3407 K299  ; 出右開夾錯誤碼
      MEP
      MOV     K3 D3409
8540  LD>=    D3407 K300  ; 出右開夾錯誤碼
      AND<=   D3407 K399  ; 出右開夾錯誤碼
      MEP
      MOV     K4 D3409
8549  LD>=    D3407 K500  ; 出右開夾錯誤碼
      AND<=   D3407 K599  ; 出右開夾錯誤碼
      MEP
      MOV     K5 D3409
8558  LD>=    D3407 K800  ; 出右開夾錯誤碼
      AND<=   D3407 K899  ; 出右開夾錯誤碼
      MEP
      MOV     K6 D3409
8567  LD>=    D3407 K900  ; 出右開夾錯誤碼
      AND<=   D3407 K999  ; 出右開夾錯誤碼
      MEP
      MOV     K7 D3409
8576  LD>=    D3407 K1200  ; 出右開夾錯誤碼
      AND<=   D3407 K1299  ; 出右開夾錯誤碼
      MEP
      MOV     K8 D3409
8585  LD>=    D3407 K2000  ; 出右開夾錯誤碼
      AND<=   D3407 K2099  ; 出右開夾錯誤碼
      MEP
      MOV     K9 D3409
8594  LDI     X0A1D  ; #14 AXIS Busy
      AND     L3482  ; 出右開夾M code ON
      MOV     D3406 D3410  ; 出右開夾M碼讀出
8598  LD<>    D3410 K0  ; 出右開夾M碼讀出
      AND     L3482  ; 出右開夾M code ON
      MOV     K1 U0A0\G5604  ; #14_M code OFF request
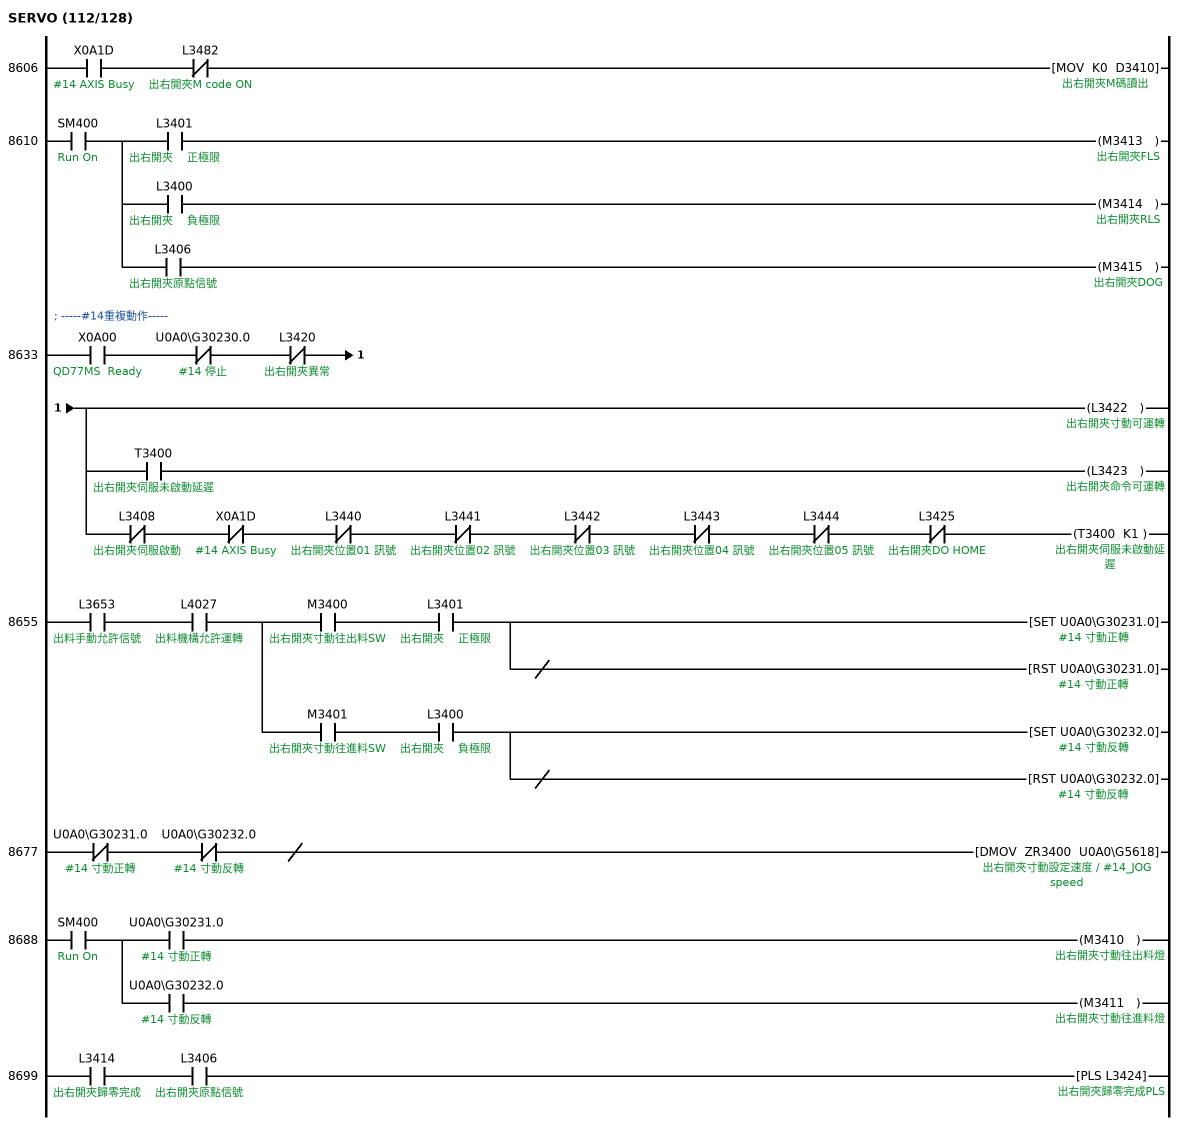
8606  LD      X0A1D  ; #14 AXIS Busy
      ANI     L3482  ; 出右開夾M code ON
      MOV     K0 D3410
8610  LD      SM400  ; Run On
      MPS
      AND     L3401  ; 出右開夾    正極限
      OUT     M3413  ; 出右開夾FLS
      MRD
      AND     L3400  ; 出右開夾    負極限
      OUT     M3414  ; 出右開夾RLS
      MPP
      AND     L3406  ; 出右開夾原點信號
      OUT     M3415  ; 出右開夾DOG
; -----#14重複動作-----
8633  LD      X0A00  ; QD77MS  Ready
      ANI     U0A0\G30230.0  ; #14 停止
      ANI     L3420  ; 出右開夾異常
      OUT     L3422  ; 出右開夾寸動可運轉
      MPS
      AND     T3400  ; 出右開夾伺服未啟動延遲
      OUT     L3423  ; 出右開夾命令可運轉
      MPP
      ANI     L3408  ; 出右開夾伺服啟動
      ANI     X0A1D  ; #14 AXIS Busy
      ANI     L3440  ; 出右開夾位置01 訊號
      ANI     L3441  ; 出右開夾位置02 訊號
      ANI     L3442  ; 出右開夾位置03 訊號
      ANI     L3443  ; 出右開夾位置04 訊號
      ANI     L3444  ; 出右開夾位置05 訊號
      ANI     L3425  ; 出右開夾DO HOME
      OUT     T3400 K1  ; 出右開夾伺服未啟動延遲
8655  LD      L3653  ; 出料手動允許信號
      AND     L4027  ; 出料機構允許運轉
      MPS
      AND     M3400  ; 出右開夾寸動往出料SW
      AND     L3401  ; 出右開夾    正極限
      SET     U0A0\G30231.0  ; #14 寸動正轉
      INV
      RST     U0A0\G30231.0  ; #14 寸動正轉
      MPP
      AND     M3401  ; 出右開夾寸動往進料SW
      AND     L3400  ; 出右開夾    負極限
      SET     U0A0\G30232.0  ; #14 寸動反轉
      INV
      RST     U0A0\G30232.0  ; #14 寸動反轉
8677  LDI     U0A0\G30231.0  ; #14 寸動正轉
      ANI     U0A0\G30232.0  ; #14 寸動反轉
      INV
      DMOV    ZR3400 U0A0\G5618  ; 出右開夾寸動設定速度 / #14_JOG     speed
8688  LD      SM400  ; Run On
      MPS
      AND     U0A0\G30231.0  ; #14 寸動正轉
      OUT     M3410  ; 出右開夾寸動往出料燈
      MPP
      AND     U0A0\G30232.0  ; #14 寸動反轉
      OUT     M3411  ; 出右開夾寸動往進料燈
8699  LD      L3414  ; 出右開夾歸零完成
      AND     L3406  ; 出右開夾原點信號
      PLS     L3424  ; 出右開夾歸零完成PLS
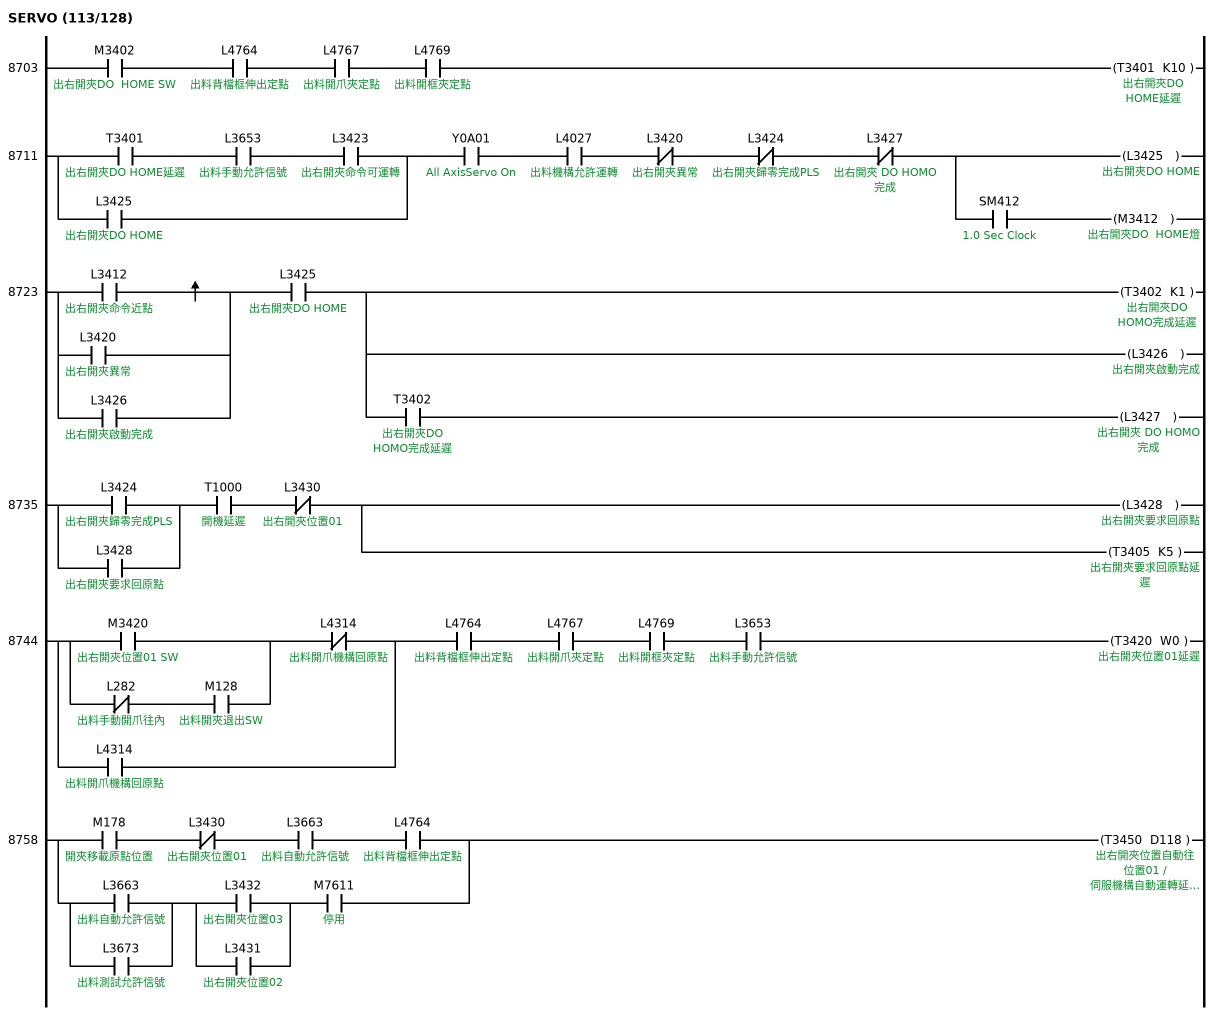
8703  LD      M3402  ; 出右開夾DO  HOME SW
      AND     L4764  ; 出料背檔框伸出定點
      AND     L4767  ; 出料開爪夾定點
      AND     L4769  ; 出料開框夾定點
      OUT     T3401 K10  ; 出右開夾DO HOME延遲
8711  LD      T3401  ; 出右開夾DO HOME延遲
      AND     L3653  ; 出料手動允許信號
      AND     L3423  ; 出右開夾命令可運轉
      OR      L3425  ; 出右開夾DO HOME
      AND     Y0A01  ; All AxisServo On
      AND     L4027  ; 出料機構允許運轉
      ANI     L3420  ; 出右開夾異常
      ANI     L3424  ; 出右開夾歸零完成PLS
      ANI     L3427  ; 出右開夾 DO HOMO 完成
      OUT     L3425  ; 出右開夾DO HOME
      AND     SM412  ; 1.0 Sec Clock
      OUT     M3412  ; 出右開夾DO  HOME燈
8723  LD      L3412  ; 出右開夾命令近點
      MEP
      OR      L3420  ; 出右開夾異常
      OR      L3426  ; 出右開夾啟動完成
      AND     L3425  ; 出右開夾DO HOME
      OUT     T3402 K1  ; 出右開夾DO HOMO完成延遲
      OUT     L3426  ; 出右開夾啟動完成
      AND     T3402  ; 出右開夾DO HOMO完成延遲
      OUT     L3427  ; 出右開夾 DO HOMO 完成
8735  LD      L3424  ; 出右開夾歸零完成PLS
      OR      L3428  ; 出右開夾要求回原點
      AND     T1000  ; 開機延遲
      ANI     L3430  ; 出右開夾位置01
      OUT     L3428  ; 出右開夾要求回原點
      OUT     T3405 K5  ; 出右開夾要求回原點延遲
8744  LD      M3420  ; 出右開夾位置01 SW
      LDI     L282  ; 出料手動開爪往內
      AND     M128  ; 出料開夾退出SW
      ORB
      ANI     L4314  ; 出料開爪機構回原點
      OR      L4314  ; 出料開爪機構回原點
      AND     L4764  ; 出料背檔框伸出定點
      AND     L4767  ; 出料開爪夾定點
      AND     L4769  ; 出料開框夾定點
      AND     L3653  ; 出料手動允許信號
      OUT     T3420 W0  ; 出右開夾位置01延遲
8758  LD      M178  ; 開夾移載原點位置
      ANI     L3430  ; 出右開夾位置01
      AND     L3663  ; 出料自動允許信號
      AND     L4764  ; 出料背檔框伸出定點
      LD      L3663  ; 出料自動允許信號
      OR      L3673  ; 出料測試允許信號
      LD      L3432  ; 出右開夾位置03
      OR      L3431  ; 出右開夾位置02
      ANB
      AND     M7611  ; 停用
      ORB
      OUT     T3450 D118  ; 出右開夾位置自動往  位置01 / 伺服機構自動運轉延遲時間
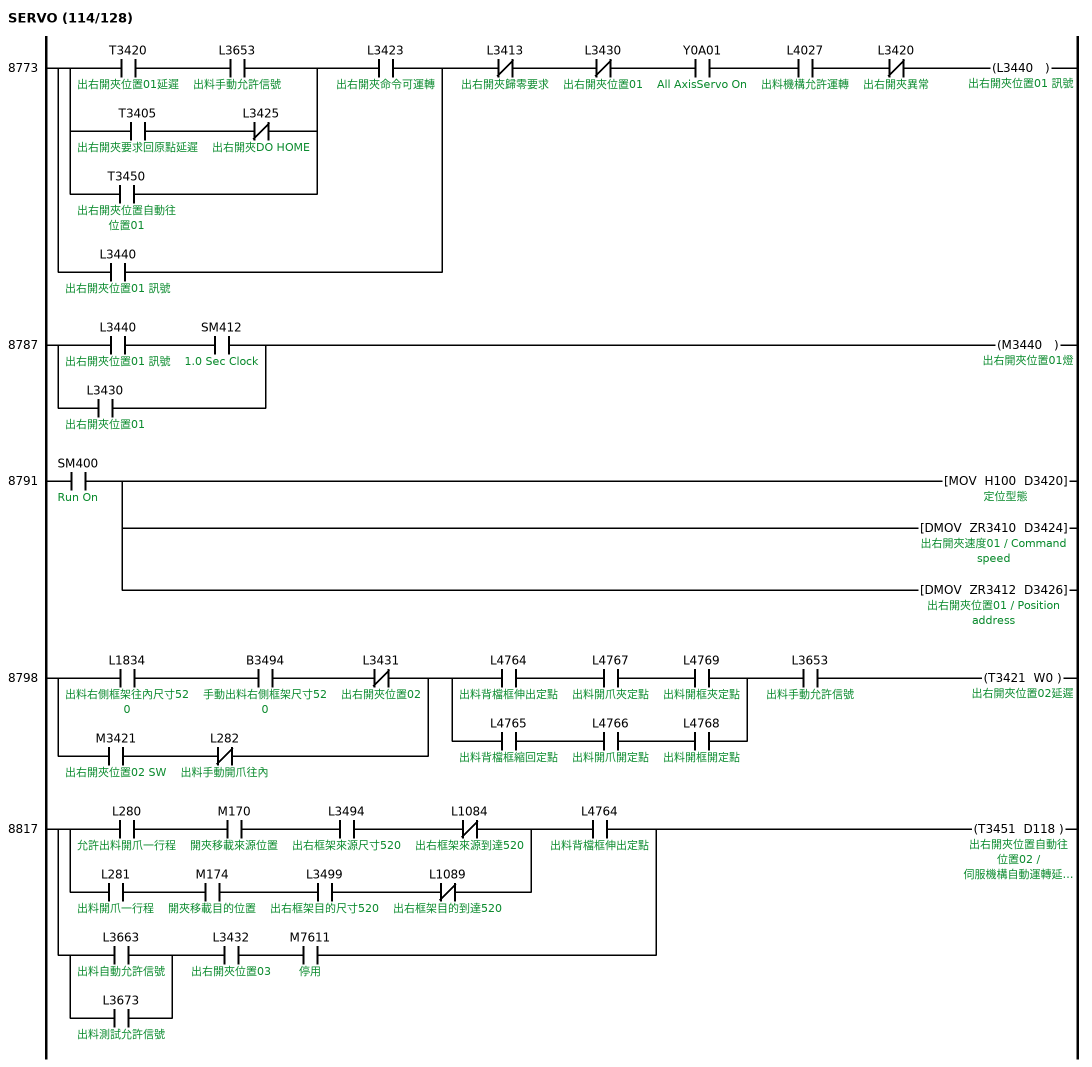
8773  LD      T3420  ; 出右開夾位置01延遲
      AND     L3653  ; 出料手動允許信號
      LD      T3405  ; 出右開夾要求回原點延遲
      ANI     L3425  ; 出右開夾DO HOME
      ORB
      OR      T3450  ; 出右開夾位置自動往  位置01
      AND     L3423  ; 出右開夾命令可運轉
      OR      L3440  ; 出右開夾位置01 訊號
      ANI     L3413  ; 出右開夾歸零要求
      ANI     L3430  ; 出右開夾位置01
      AND     Y0A01  ; All AxisServo On
      AND     L4027  ; 出料機構允許運轉
      ANI     L3420  ; 出右開夾異常
      OUT     L3440  ; 出右開夾位置01 訊號
8787  LD      L3440  ; 出右開夾位置01 訊號
      AND     SM412  ; 1.0 Sec Clock
      OR      L3430  ; 出右開夾位置01
      OUT     M3440  ; 出右開夾位置01燈
8791  LD      SM400  ; Run On
      MOV     H100 D3420  ; 定位型態
      DMOV    ZR3410 D3424  ; 出右開夾速度01 / Command  speed
      DMOV    ZR3412 D3426  ; Position address
8798  LD      L1834  ; 出料右側框架往內尺寸520
      AND     B3494  ; 手動出料右側框架尺寸520
      ANI     L3431  ; 出右開夾位置02
      LD      M3421  ; 出右開夾位置02 SW
      ANI     L282  ; 出料手動開爪往內
      ORB
      LD      L4764  ; 出料背檔框伸出定點
      AND     L4767  ; 出料開爪夾定點
      AND     L4769  ; 出料開框夾定點
      LD      L4765  ; 出料背檔框縮回定點
      AND     L4766  ; 出料開爪開定點
      AND     L4768  ; 出料開框開定點
      ORB
      ANB
      AND     L3653  ; 出料手動允許信號
      OUT     T3421 W0  ; 出右開夾位置02延遲
8817  LD      L280  ; 允許出料開爪一行程
      AND     M170  ; 開夾移載來源位置
      AND     L3494  ; 出右框架來源尺寸520
      ANI     L1084  ; 出右框架來源到達520
      LD      L281  ; 出料開爪一行程
      AND     M174  ; 開夾移載目的位置
      AND     L3499  ; 出右框架目的尺寸520
      ANI     L1089  ; 出右框架目的到達520
      ORB
      AND     L4764  ; 出料背檔框伸出定點
      LD      L3663  ; 出料自動允許信號
      OR      L3673  ; 出料測試允許信號
      AND     L3432  ; 出右開夾位置03
      AND     M7611  ; 停用
      ORB
      OUT     T3451 D118  ; 出右開夾位置自動往  位置02 / 伺服機構自動運轉延遲時間
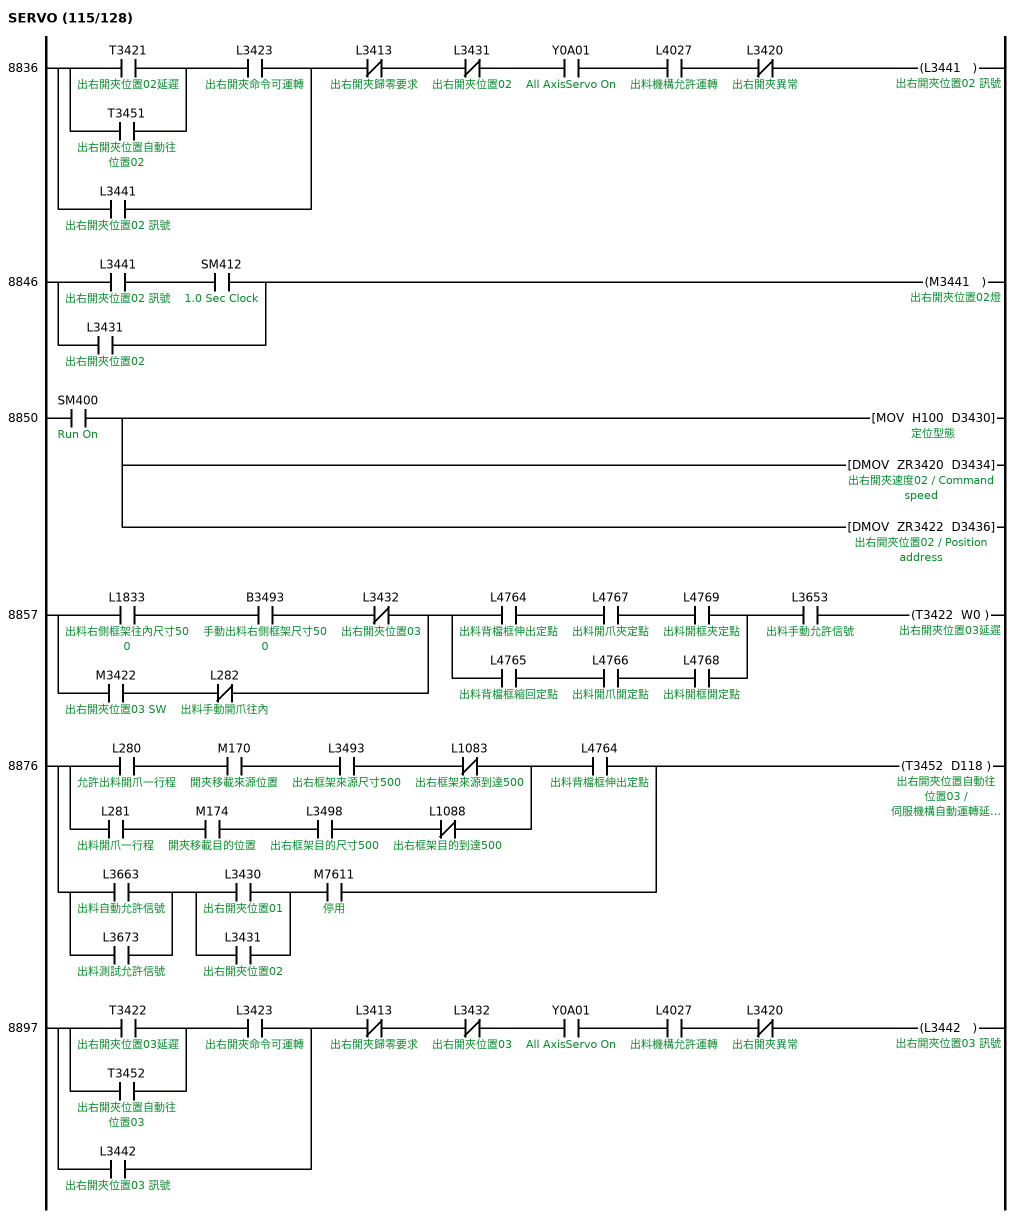
8836  LD      T3421  ; 出右開夾位置02延遲
      OR      T3451  ; 出右開夾位置自動往  位置02
      AND     L3423  ; 出右開夾命令可運轉
      OR      L3441  ; 出右開夾位置02 訊號
      ANI     L3413  ; 出右開夾歸零要求
      ANI     L3431  ; 出右開夾位置02
      AND     Y0A01  ; All AxisServo On
      AND     L4027  ; 出料機構允許運轉
      ANI     L3420  ; 出右開夾異常
      OUT     L3441  ; 出右開夾位置02 訊號
8846  LD      L3441  ; 出右開夾位置02 訊號
      AND     SM412  ; 1.0 Sec Clock
      OR      L3431  ; 出右開夾位置02
      OUT     M3441  ; 出右開夾位置02燈
8850  LD      SM400  ; Run On
      MOV     H100 D3430  ; 定位型態
      DMOV    ZR3420 D3434  ; 出右開夾速度02 / Command  speed
      DMOV    ZR3422 D3436  ; Position address
8857  LD      L1833  ; 出料右側框架往內尺寸500
      AND     B3493  ; 手動出料右側框架尺寸500
      ANI     L3432  ; 出右開夾位置03
      LD      M3422  ; 出右開夾位置03 SW
      ANI     L282  ; 出料手動開爪往內
      ORB
      LD      L4764  ; 出料背檔框伸出定點
      AND     L4767  ; 出料開爪夾定點
      AND     L4769  ; 出料開框夾定點
      LD      L4765  ; 出料背檔框縮回定點
      AND     L4766  ; 出料開爪開定點
      AND     L4768  ; 出料開框開定點
      ORB
      ANB
      AND     L3653  ; 出料手動允許信號
      OUT     T3422 W0  ; 出右開夾位置03延遲
8876  LD      L280  ; 允許出料開爪一行程
      AND     M170  ; 開夾移載來源位置
      AND     L3493  ; 出右框架來源尺寸500
      ANI     L1083  ; 出右框架來源到達500
      LD      L281  ; 出料開爪一行程
      AND     M174  ; 開夾移載目的位置
      AND     L3498  ; 出右框架目的尺寸500
      ANI     L1088  ; 出右框架目的到達500
      ORB
      AND     L4764  ; 出料背檔框伸出定點
      LD      L3663  ; 出料自動允許信號
      OR      L3673  ; 出料測試允許信號
      LD      L3430  ; 出右開夾位置01
      OR      L3431  ; 出右開夾位置02
      ANB
      AND     M7611  ; 停用
      ORB
      OUT     T3452 D118  ; 出右開夾位置自動往  位置03 / 伺服機構自動運轉延遲時間
8897  LD      T3422  ; 出右開夾位置03延遲
      OR      T3452  ; 出右開夾位置自動往  位置03
      AND     L3423  ; 出右開夾命令可運轉
      OR      L3442  ; 出右開夾位置03 訊號
      ANI     L3413  ; 出右開夾歸零要求
      ANI     L3432  ; 出右開夾位置03
      AND     Y0A01  ; All AxisServo On
      AND     L4027  ; 出料機構允許運轉
      ANI     L3420  ; 出右開夾異常
      OUT     L3442  ; 出右開夾位置03 訊號
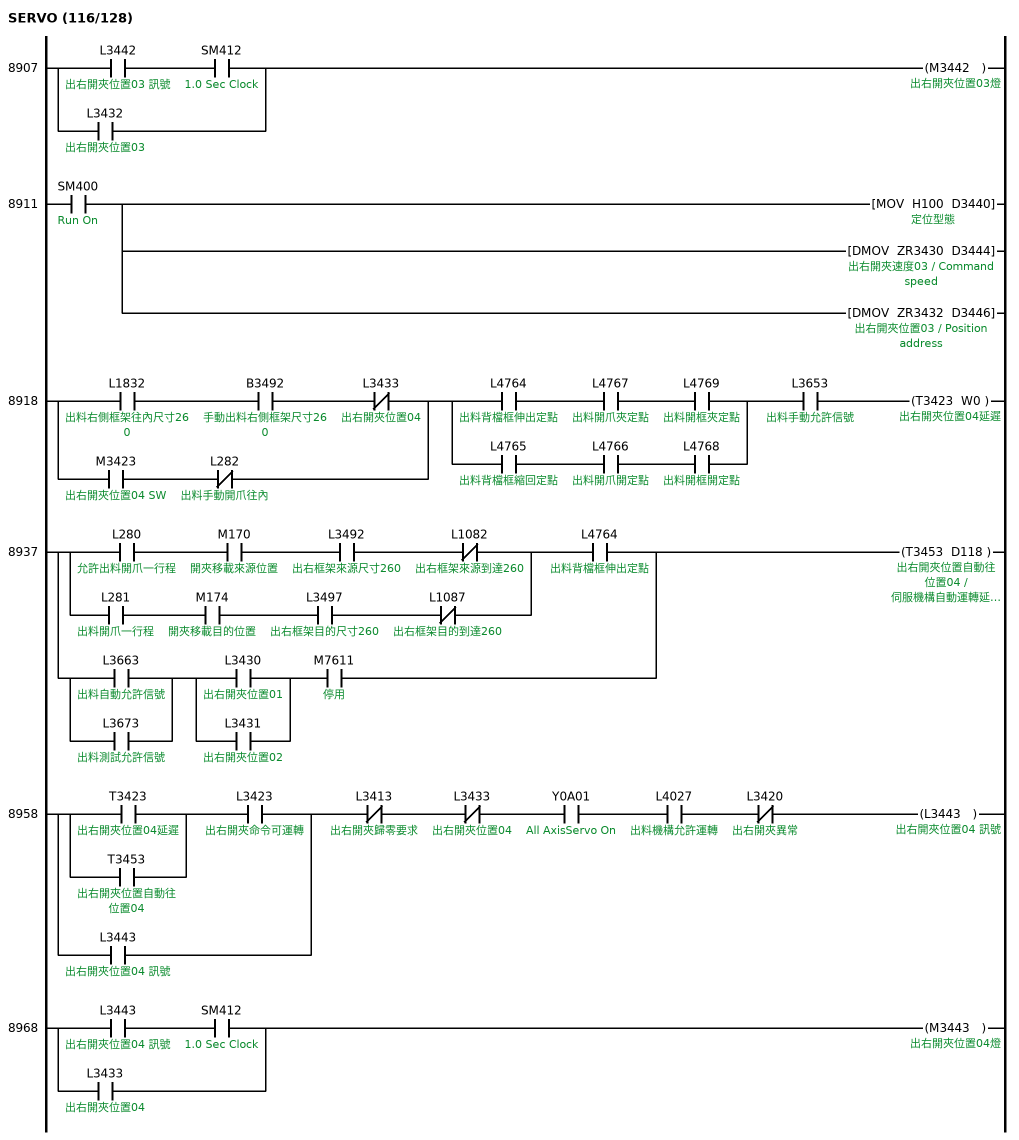
8907  LD      L3442  ; 出右開夾位置03 訊號
      AND     SM412  ; 1.0 Sec Clock
      OR      L3432  ; 出右開夾位置03
      OUT     M3442  ; 出右開夾位置03燈
8911  LD      SM400  ; Run On
      MOV     H100 D3440  ; 定位型態
      DMOV    ZR3430 D3444  ; 出右開夾速度03 / Command  speed
      DMOV    ZR3432 D3446  ; Position address
8918  LD      L1832  ; 出料右側框架往內尺寸260
      AND     B3492  ; 手動出料右側框架尺寸260
      ANI     L3433  ; 出右開夾位置04
      LD      M3423  ; 出右開夾位置04 SW
      ANI     L282  ; 出料手動開爪往內
      ORB
      LD      L4764  ; 出料背檔框伸出定點
      AND     L4767  ; 出料開爪夾定點
      AND     L4769  ; 出料開框夾定點
      LD      L4765  ; 出料背檔框縮回定點
      AND     L4766  ; 出料開爪開定點
      AND     L4768  ; 出料開框開定點
      ORB
      ANB
      AND     L3653  ; 出料手動允許信號
      OUT     T3423 W0  ; 出右開夾位置04延遲
8937  LD      L280  ; 允許出料開爪一行程
      AND     M170  ; 開夾移載來源位置
      AND     L3492  ; 出右框架來源尺寸260
      ANI     L1082  ; 出右框架來源到達260
      LD      L281  ; 出料開爪一行程
      AND     M174  ; 開夾移載目的位置
      AND     L3497  ; 出右框架目的尺寸260
      ANI     L1087  ; 出右框架目的到達260
      ORB
      AND     L4764  ; 出料背檔框伸出定點
      LD      L3663  ; 出料自動允許信號
      OR      L3673  ; 出料測試允許信號
      LD      L3430  ; 出右開夾位置01
      OR      L3431  ; 出右開夾位置02
      ANB
      AND     M7611  ; 停用
      ORB
      OUT     T3453 D118  ; 出右開夾位置自動往  位置04 / 伺服機構自動運轉延遲時間
8958  LD      T3423  ; 出右開夾位置04延遲
      OR      T3453  ; 出右開夾位置自動往  位置04
      AND     L3423  ; 出右開夾命令可運轉
      OR      L3443  ; 出右開夾位置04 訊號
      ANI     L3413  ; 出右開夾歸零要求
      ANI     L3433  ; 出右開夾位置04
      AND     Y0A01  ; All AxisServo On
      AND     L4027  ; 出料機構允許運轉
      ANI     L3420  ; 出右開夾異常
      OUT     L3443  ; 出右開夾位置04 訊號
8968  LD      L3443  ; 出右開夾位置04 訊號
      AND     SM412  ; 1.0 Sec Clock
      OR      L3433  ; 出右開夾位置04
      OUT     M3443  ; 出右開夾位置04燈
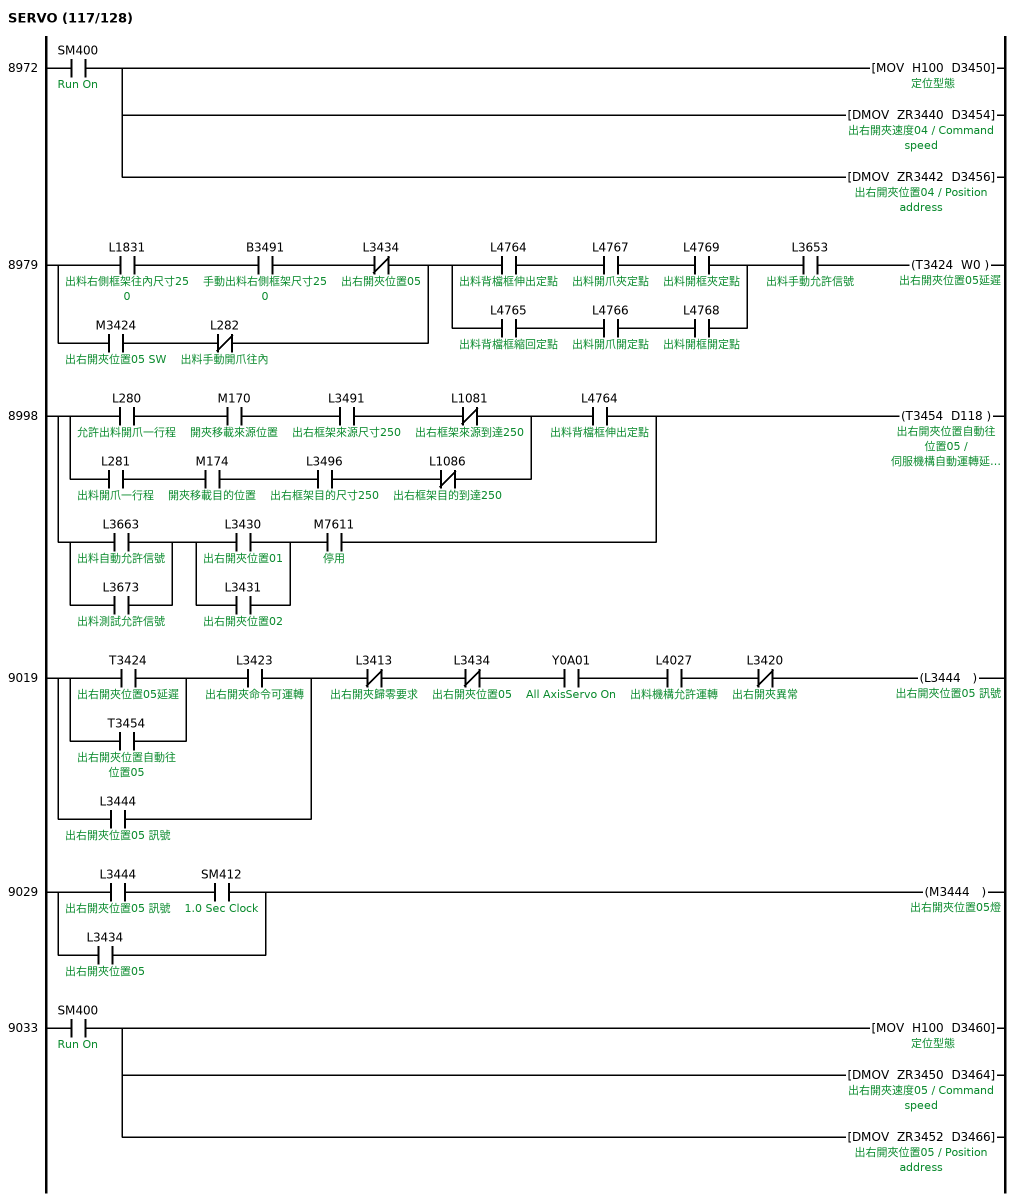
8972  LD      SM400  ; Run On
      MOV     H100 D3450  ; 定位型態
      DMOV    ZR3440 D3454  ; 出右開夾速度04 / Command  speed
      DMOV    ZR3442 D3456  ; Position address
8979  LD      L1831  ; 出料右側框架往內尺寸250
      AND     B3491  ; 手動出料右側框架尺寸250
      ANI     L3434  ; 出右開夾位置05
      LD      M3424  ; 出右開夾位置05 SW
      ANI     L282  ; 出料手動開爪往內
      ORB
      LD      L4764  ; 出料背檔框伸出定點
      AND     L4767  ; 出料開爪夾定點
      AND     L4769  ; 出料開框夾定點
      LD      L4765  ; 出料背檔框縮回定點
      AND     L4766  ; 出料開爪開定點
      AND     L4768  ; 出料開框開定點
      ORB
      ANB
      AND     L3653  ; 出料手動允許信號
      OUT     T3424 W0  ; 出右開夾位置05延遲
8998  LD      L280  ; 允許出料開爪一行程
      AND     M170  ; 開夾移載來源位置
      AND     L3491  ; 出右框架來源尺寸250
      ANI     L1081  ; 出右框架來源到達250
      LD      L281  ; 出料開爪一行程
      AND     M174  ; 開夾移載目的位置
      AND     L3496  ; 出右框架目的尺寸250
      ANI     L1086  ; 出右框架目的到達250
      ORB
      AND     L4764  ; 出料背檔框伸出定點
      LD      L3663  ; 出料自動允許信號
      OR      L3673  ; 出料測試允許信號
      LD      L3430  ; 出右開夾位置01
      OR      L3431  ; 出右開夾位置02
      ANB
      AND     M7611  ; 停用
      ORB
      OUT     T3454 D118  ; 出右開夾位置自動往  位置05 / 伺服機構自動運轉延遲時間
9019  LD      T3424  ; 出右開夾位置05延遲
      OR      T3454  ; 出右開夾位置自動往  位置05
      AND     L3423  ; 出右開夾命令可運轉
      OR      L3444  ; 出右開夾位置05 訊號
      ANI     L3413  ; 出右開夾歸零要求
      ANI     L3434  ; 出右開夾位置05
      AND     Y0A01  ; All AxisServo On
      AND     L4027  ; 出料機構允許運轉
      ANI     L3420  ; 出右開夾異常
      OUT     L3444  ; 出右開夾位置05 訊號
9029  LD      L3444  ; 出右開夾位置05 訊號
      AND     SM412  ; 1.0 Sec Clock
      OR      L3434  ; 出右開夾位置05
      OUT     M3444  ; 出右開夾位置05燈
9033  LD      SM400  ; Run On
      MOV     H100 D3460  ; 定位型態
      DMOV    ZR3450 D3464  ; 出右開夾速度05 / Command  speed
      DMOV    ZR3452 D3466  ; Position address
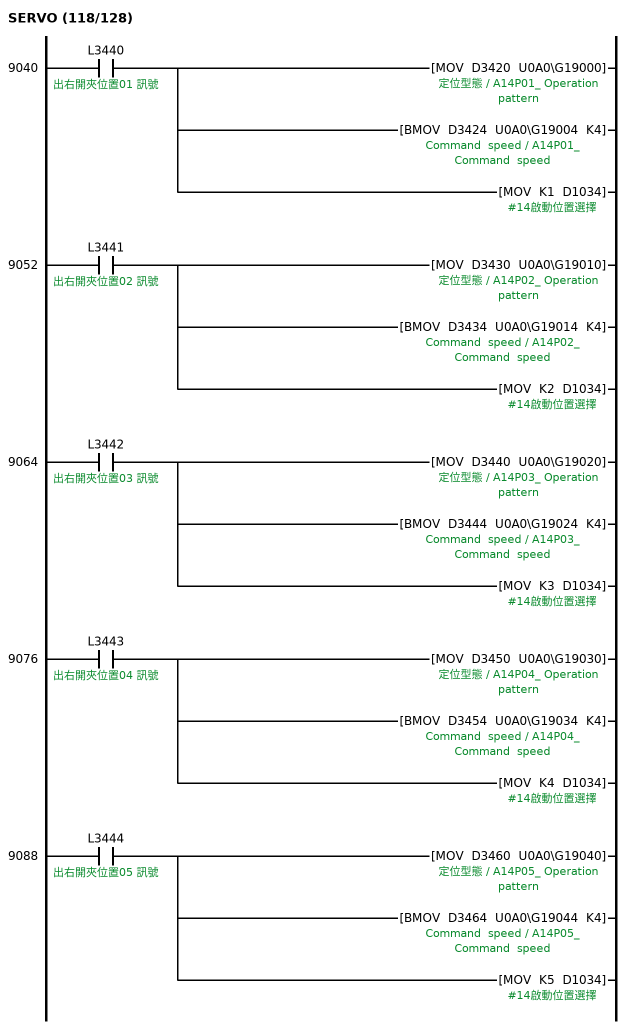
9040  LD      L3440  ; 出右開夾位置01 訊號
      MOV     D3420 U0A0\G19000  ; A14P01_ Operation pattern
      BMOV    D3424 U0A0\G19004 K4  ; A14P01_ Command  speed
      MOV     K1 D1034  ; #14啟動位置選擇
9052  LD      L3441  ; 出右開夾位置02 訊號
      MOV     D3430 U0A0\G19010  ; A14P02_ Operation pattern
      BMOV    D3434 U0A0\G19014 K4  ; A14P02_ Command  speed
      MOV     K2 D1034
9064  LD      L3442  ; 出右開夾位置03 訊號
      MOV     D3440 U0A0\G19020  ; A14P03_ Operation pattern
      BMOV    D3444 U0A0\G19024 K4  ; A14P03_ Command  speed
      MOV     K3 D1034
9076  LD      L3443  ; 出右開夾位置04 訊號
      MOV     D3450 U0A0\G19030  ; A14P04_ Operation pattern
      BMOV    D3454 U0A0\G19034 K4  ; A14P04_ Command  speed
      MOV     K4 D1034
9088  LD      L3444  ; 出右開夾位置05 訊號
      MOV     D3460 U0A0\G19040  ; A14P05_ Operation pattern
      BMOV    D3464 U0A0\G19044 K4  ; A14P05_ Command  speed
      MOV     K5 D1034
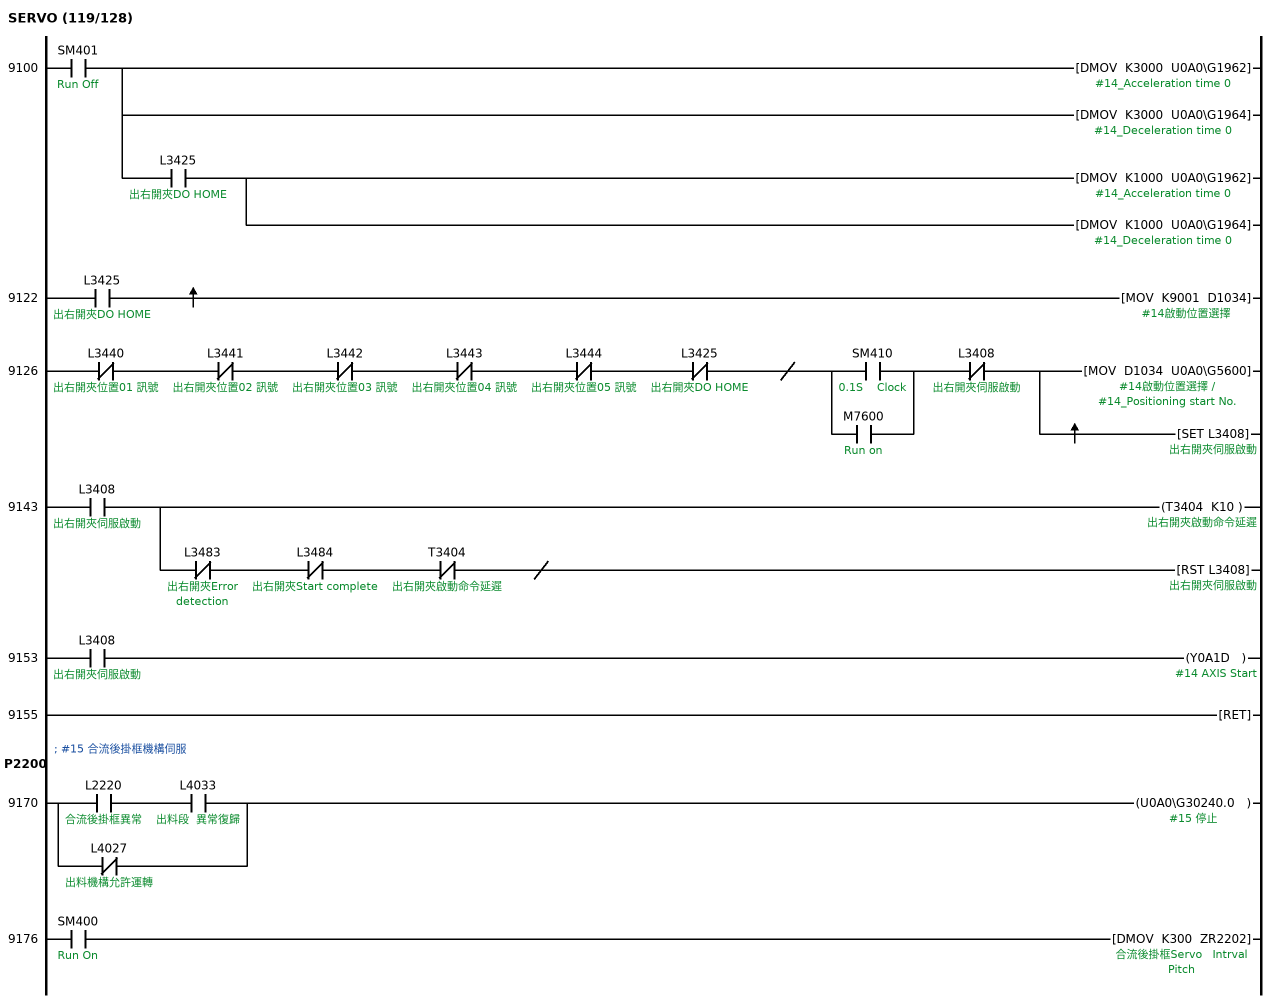
9100  LD      SM401  ; Run Off
      DMOV    K3000 U0A0\G1962  ; #14_Acceleration time 0
      DMOV    K3000 U0A0\G1964  ; #14_Deceleration time 0
      AND     L3425  ; 出右開夾DO HOME
      DMOV    K1000 U0A0\G1962
      DMOV    K1000 U0A0\G1964
9122  LD      L3425  ; 出右開夾DO HOME
      MEP
      MOV     K9001 D1034
9126  LDI     L3440  ; 出右開夾位置01 訊號
      ANI     L3441  ; 出右開夾位置02 訊號
      ANI     L3442  ; 出右開夾位置03 訊號
      ANI     L3443  ; 出右開夾位置04 訊號
      ANI     L3444  ; 出右開夾位置05 訊號
      ANI     L3425  ; 出右開夾DO HOME
      INV
      LD      SM410  ; 0.1S    Clock
      OR      M7600  ; Run on
      ANB
      ANI     L3408  ; 出右開夾伺服啟動
      MOV     D1034 U0A0\G5600  ; #14_Positioning start No.
      MEP
      SET     L3408  ; 出右開夾伺服啟動
9143  LD      L3408  ; 出右開夾伺服啟動
      OUT     T3404 K10  ; 出右開夾啟動命令延遲
      ANI     L3483  ; 出右開夾Error detection
      ANI     L3484  ; 出右開夾Start complete
      ANI     T3404  ; 出右開夾啟動命令延遲
      INV
      RST     L3408  ; 出右開夾伺服啟動
9153  LD      L3408  ; 出右開夾伺服啟動
      OUT     Y0A1D  ; #14 AXIS Start
9155  RET
; #15 合流後掛框機構伺服
      P2200
9170  LD      L2220  ; 合流後掛框異常
      AND     L4033  ; 出料段  異常復歸
      ORI     L4027  ; 出料機構允許運轉
      OUT     U0A0\G30240.0  ; #15 停止
9176  LD      SM400  ; Run On
      DMOV    K300 ZR2202  ; 合流後掛框Servo   Intrval Pitch
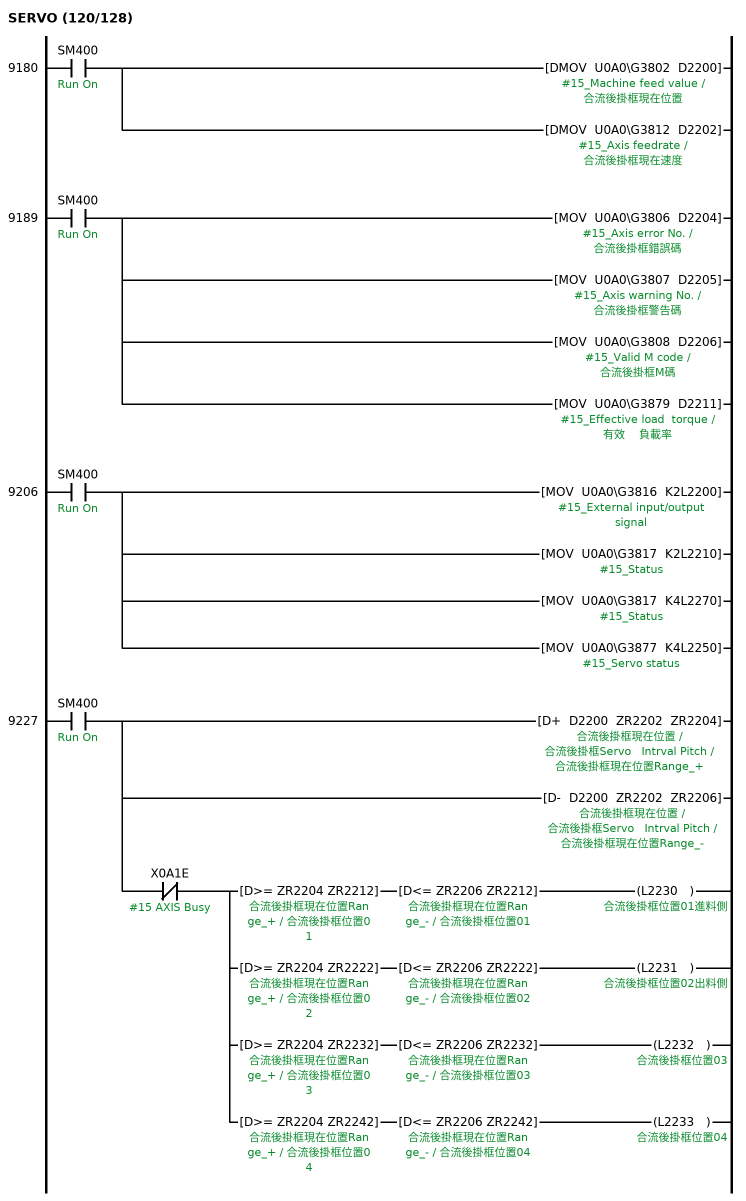
9180  LD      SM400  ; Run On
      DMOV    U0A0\G3802 D2200  ; #15_Machine feed value / 合流後掛框現在位置
      DMOV    U0A0\G3812 D2202  ; #15_Axis feedrate / 合流後掛框現在速度
9189  LD      SM400  ; Run On
      MOV     U0A0\G3806 D2204  ; #15_Axis error No. / 合流後掛框錯誤碼
      MOV     U0A0\G3807 D2205  ; #15_Axis warning No. / 合流後掛框警告碼
      MOV     U0A0\G3808 D2206  ; #15_Valid M code / 合流後掛框M碼
      MOV     U0A0\G3879 D2211  ; #15_Effective load  torque / 有效    負載率
9206  LD      SM400  ; Run On
      MOV     U0A0\G3816 K2L2200  ; #15_External input/output signal / 合流後掛框    負極限
      MOV     U0A0\G3817 K2L2210  ; #15_Status / 合流後掛框速度控制
      MOV     U0A0\G3817 K4L2270  ; 合流後掛框速度控制
      MOV     U0A0\G3877 K4L2250  ; #15_Servo status / READY ON
9227  LD      SM400  ; Run On
      D+      D2200 ZR2202 ZR2204  ; 合流後掛框現在位置Range_+
      D-      D2200 ZR2202 ZR2206  ; 合流後掛框現在位置Range_-
      ANI     X0A1E  ; #15 AXIS Busy
      MPS
      ANDD>=  ZR2204 ZR2212  ; 合流後掛框現在位置Range_+ / 合流後掛框位置01
      ANDD<=  ZR2206 ZR2212  ; 合流後掛框現在位置Range_- / 合流後掛框位置01
      OUT     L2230  ; 合流後掛框位置01進料側
      MRD
      ANDD>=  ZR2204 ZR2222  ; 合流後掛框現在位置Range_+ / 合流後掛框位置02
      ANDD<=  ZR2206 ZR2222  ; 合流後掛框現在位置Range_- / 合流後掛框位置02
      OUT     L2231  ; 合流後掛框位置02出料側
      MRD
      ANDD>=  ZR2204 ZR2232  ; 合流後掛框現在位置Range_+ / 合流後掛框位置03
      ANDD<=  ZR2206 ZR2232  ; 合流後掛框現在位置Range_- / 合流後掛框位置03
      OUT     L2232  ; 合流後掛框位置03
      MPP
      ANDD>=  ZR2204 ZR2242  ; 合流後掛框現在位置Range_+ / 合流後掛框位置04
      ANDD<=  ZR2206 ZR2242  ; 合流後掛框現在位置Range_- / 合流後掛框位置04
      OUT     L2233  ; 合流後掛框位置04
